Omron CX-Programmer project IO_TEST (CX-Programmer 9.20)

# PLC ELT215PLC: C200HE CPU42

## Global symbols (name address type ; comment)
0.00 BOOL  ; T_OUTPUT_FRONT GATE CLOSE
0.01 BOOL  ; T_OUTPUT_PULL IN PART
0.02 BOOL  ; T_OUTPUT_CLAMP ENGAGE
0.03 BOOL  ; T_OUTPUT_ALIGNMENT CLAMP RETRACT
0.04 BOOL  ; T_OUTPUT_TURNTABLE ROTATE FORWARD
0.05 BOOL  ; T_OUTPUT_EXIT GATE OPEN
0.06 BOOL  ; T_OUTPUT_DC_TEST_OUT
0.07 BOOL  ; T_OUTPUT_START SEQUENCER
0.08 BOOL  ; T_OUTPUT_BUZZER (INTERMITTENT)
0.09 BOOL  ; T_OUTPUT_PUSH OUT PART
0.10 BOOL  ; F_OUTPUT_FEED1 EXTEND
0.11 BOOL  ; F_OUTPUT_FEED2 EXTEND
0.12 BOOL  ; --== DO NOT USE ==--
0.13 BOOL  ; --== DO NOT USE ==--
0.14 BOOL  ; --== DO NOT USE ==--
0.15 BOOL  ; --== DO NOT USE ==--
1.00 BOOL  ; T_OUTPUT_THIRD TIME RELAY
1.01 BOOL  ; ID_OUTPUT_FRONT GATE CLOSE
1.02 BOOL  ; ID_OUTPUT_PUSH IN
1.03 BOOL  ; ID_OUTPUT_CLAMP ENGAGE
1.04 BOOL  ; ID_OUTPUT_TRAP DOOR OPEN
1.05 BOOL  ; ID_OUTPUT_PUSH OUT AND ELEVATE AND BACK GATE OPEN
1.06 BOOL  ; Output #6, Block 2 UNUSED
1.07 BOOL  ; ID_OUTPUT_JURASSIC GATE PULL UP
1.08 BOOL  ; --== DO NOT USE ==--
1.09 BOOL  ; --== DO NOT USE ==--
1.10 BOOL  ; --== DO NOT USE ==--
1.11 BOOL  ; --== DO NOT USE ==--
1.12 BOOL  ; --== DO NOT USE ==--
1.13 BOOL  ; --== DO NOT USE ==--
1.14 BOOL  ; --== DO NOT USE ==--
1.15 BOOL  ; --== DO NOT USE ==--
232.00 BOOL  ; F_WB_FEED1 EXTEND ONESHOT
232.01 BOOL  ; F_WB_FEED2 EXTEND ONESHOT
232.02 BOOL  ; F_WB_SEQUENCE RUNNING LATCH
232.03 BOOL  ; F_WB_FEEDER 1 PARTS EXTENSION PULSES
232.04 BOOL  ; F_WB_FEEDER 2 PARTS EXTENSION PULSES
232.05 BOOL  ; F_UNUSED WORK BIT
232.06 BOOL  ; F_UNUSED WORK BIT
232.07 BOOL  ; F_UNUSED WORK BIT
232.08 BOOL  ; F_UNUSED WORK BIT
232.09 BOOL  ; F_UNUSED WORK BIT
232.10 BOOL  ; F_UNUSED WORK BIT
232.11 BOOL  ; F_UNUSED WORK BIT
232.12 BOOL  ; F_UNUSED WORK BIT
232.13 BOOL  ; F_UNUSED WORK BIT
232.14 BOOL  ; F_UNUSED WORK BIT
232.15 BOOL  ; F_UNUSED WORK BIT
233.00 BOOL  ; F_UNUSED WORK BIT
233.01 BOOL  ; F_WB_PART 1 TIMER SILENCER
233.02 BOOL  ; F_WB_PART 2 TIMER SILENCER
233.03 BOOL  ; F_WB_PART 3 TIMER SILENCER
233.04 BOOL  ; F_WB_PART 4 TIMER SILENCER
233.05 BOOL  ; F_WB_PART 5 TIMER SILENCER
233.06 BOOL  ; F_WB_PART 6 TIMER SILENCER
233.07 BOOL  ; F_WB_PART 7 TIMER SILENCER
233.08 BOOL  ; F_WB_PART 8 TIMER SILENCER
233.09 BOOL  ; F_WB_PART 9 TIMER SILENCER
233.10 BOOL  ; F_WB_PART 10 TIMER SILENCER
233.11 BOOL  ; F_UNUSED WORK BIT
233.12 BOOL  ; F_UNUSED WORK BIT
233.13 BOOL  ; F_UNUSED WORK BIT
233.14 BOOL  ; F_UNUSED WORK BIT
233.15 BOOL  ; F_UNUSED WORK BIT
234.00 BOOL  ; F_UNUSED WORK BIT
234.01 BOOL  ; F_UNUSED WORK BIT
234.02 BOOL  ; F_UNUSED WORK BIT
234.03 BOOL  ; F_UNUSED WORK BIT
234.04 BOOL  ; F_UNUSED WORK BIT
234.05 BOOL  ; F_UNUSED WORK BIT
234.06 BOOL  ; F_UNUSED WORK BIT
234.07 BOOL  ; F_UNUSED WORK BIT
234.08 BOOL  ; F_UNUSED WORK BIT
234.09 BOOL  ; F_UNUSED WORK BIT
234.10 BOOL  ; F_UNUSED WORK BIT
234.11 BOOL  ; F_UNUSED WORK BIT
234.12 BOOL  ; F_UNUSED WORK BIT
234.13 BOOL  ; F_UNUSED WORK BIT
234.14 BOOL  ; F_UNUSED WORK BIT
234.15 BOOL  ; F_UNUSED WORK BIT
235.00 BOOL  ; F_UNUSED WORK BIT
235.01 BOOL  ; F_UNUSED WORK BIT
235.02 BOOL  ; F_UNUSED WORK BIT
235.03 BOOL  ; F_UNUSED WORK BIT
235.04 BOOL  ; F_UNUSED WORK BIT
235.05 BOOL  ; F_UNUSED WORK BIT
235.06 BOOL  ; F_UNUSED WORK BIT
235.07 BOOL  ; F_UNUSED WORK BIT
235.08 BOOL  ; F_UNUSED WORK BIT
235.09 BOOL  ; F_UNUSED WORK BIT
235.10 BOOL  ; F_UNUSED WORK BIT
235.11 BOOL  ; F_UNUSED WORK BIT
235.12 BOOL  ; F_UNUSED WORK BIT
235.13 BOOL  ; F_UNUSED WORK BIT
235.14 BOOL  ; F_UNUSED WORK BIT
235.15 BOOL  ; F_UNUSED WORK BIT
2.00 BOOL  ; T_INPUT_HSS
2.01 BOOL  ; T_INPUT_LSS
2.02 BOOL  ; T_INPUT_PAG SENSOR
2.03 BOOL  ; T_INPUT_TESTING STATION EMERGENCY HOME
2.04 BOOL  ; Input #4 Block 3
2.05 BOOL  ; ALL_INPUT_EMERGENCY HOME
2.06 BOOL  ; Input #6 Block 3
2.07 BOOL  ; F_INPUT_START FEEDER SEQUENCE
2.08 BOOL  ; F_INPUT_STOP FEEDER SEQUENCE
2.09 BOOL  ; Input #9 Block 3
2.10 BOOL  ; ID_INPUT_ID STATION EMERGENCY HOME
2.11 BOOL  ; ID_INPUT_IR PROXIMITY SENSOR
2.12 BOOL  ; ID_INPUT_THRU BEAM SENSOR
2.13 BOOL  ; ID_INPUT_ULTRASONIC SENSOR
2.14 BOOL  ; ID_INPUT_INDUCTIVE SENSOR
2.15 BOOL  ; ID_INPUT_PPG SENSOR
310.00 BOOL  ; T_WB_NEED HOLD FOR TESTING 1
310.01 BOOL  ; T_WB_NEED TO REORIENT 1
310.02 BOOL  ; T_NEED TO ABORT 1
310.03 BOOL  ; T_WB_NEED HOLD FOR TESTING 2
310.04 BOOL  ; T_WB_NEED TO REORIENT 2
310.05 BOOL  ; T_WB_NEED TO ABORT 2
310.06 BOOL  ; T_WB_LOCKED FRONT GATE CYLINDER LATCH
310.07 BOOL  ; T_WB_NEW PART AT GATE ONESHOT
310.08 BOOL  ; T_WB_NEW PAG DELAYED ONESHOT
310.09 BOOL  ; T_WB_PULL IN PART TRIG
310.10 BOOL  ; T_WB_LOCK FRONT GATE TRIG
310.11 BOOL  ; T_WB_RESEAT PART TRIG
310.12 BOOL  ; T_PULL IN TIMING ONESHOT
310.13 BOOL  ; T_WB_UNLOCK FRONT GATE TRIG
310.14 BOOL  ; T_WB_SEQ START PULSE
310.15 BOOL  ; T_WB_SEQ START DELAY LATCH
311.00 BOOL  ; T_WB_ABORT PROGRAM TRIG
311.01 BOOL  ; T_WB_T104 DRIVER
311.02 BOOL  ; T_WB_PART IN STATION LATCH
311.03 BOOL  ; T_WB_UNCLAMP
311.04 BOOL  ; T_WB_CLAMP
311.05 BOOL  ; T_WB_CLAMPED
311.06 BOOL  ; T_WB_ABORTING
311.07 BOOL  ; T_WB_REORIENTING
311.08 BOOL  ; T_WB_HOLDING FOR TEST
311.09 BOOL  ; T_WB_REORIENT DONE
311.10 BOOL  ; T_WB_ROTATE FORWARD DONE
311.11 BOOL  ; T_WB_ROTATE FORWARD WORKBIT
311.12 BOOL  ; T_WB_BUZZER ANNOUNCEMENT STATE
311.13 BOOL  ; T_WB_REORIENT UNCLAMP LENGTH PULSE
311.14 BOOL  ; T_WB_RESEATING PUSH DONE
311.15 BOOL  ; T_WB_RETRACT ALIGNMENT CLAMP
312.00 BOOL  ; T_WB_BACKWARDS ROTATION COMPLETE
312.01 BOOL  ; T_WB_LED TESTING STATE
312.02 BOOL  ; T_WB_DONE WITH TEST
312.03 BOOL  ; T_WB_DONE WITH TEST UNCLAMP PULSE LENGTH
312.04 BOOL  ; T_WB_READY FOR PUSH OUT
312.05 BOOL  ; T_WB_PUSHING OUT
312.06 BOOL  ; T_WB_OPEN EXIT GATE
312.07 BOOL  ; T_WB_T117 DRIVER
312.08 BOOL  ; T_WB_PLACEHOLDER
312.09 BOOL  ; T_WB_USED TO BE 0dot01 PULL IN PART
312.10 BOOL  ; T_WB_INITITAL PULL COMMAND LATCH
312.11 BOOL  ; T_WB_RESEAT PULL LATCH
312.12 BOOL  ; T_WB_USED TO BE PULL IN PART TRIG 310dot09
312.13 BOOL  ; T_WB_USED TO BE RESEAT PART TRIG 310dot11
312.14 BOOL  ; T_UNUSED WORK BIT
312.15 BOOL  ; T_UNUSED WORK BIT
313.00 BOOL  ; T_UNUSED WORK BIT
313.01 BOOL  ; T_UNUSED WORK BIT
313.02 BOOL  ; T_UNUSED WORK BIT
313.03 BOOL  ; T_UNUSED WORK BIT
313.04 BOOL  ; T_UNUSED WORK BIT
313.05 BOOL  ; T_UNUSED WORK BIT
313.06 BOOL  ; T_UNUSED WORK BIT
313.07 BOOL  ; T_UNUSED WORK BIT
313.08 BOOL  ; T_UNUSED WORK BIT
313.09 BOOL  ; T_UNUSED WORK BIT
313.10 BOOL  ; T_UNUSED WORK BIT
313.11 BOOL  ; T_UNUSED WORK BIT
313.12 BOOL  ; T_UNUSED WORK BIT
313.13 BOOL  ; T_UNUSED WORK BIT
313.14 BOOL  ; T_UNUSED WORK BIT
313.15 BOOL  ; T_UNUSED WORK BIT
314.00 BOOL  ; T_UNUSED WORK BIT
314.01 BOOL  ; T_UNUSED WORK BIT
314.02 BOOL  ; T_UNUSED WORK BIT
314.03 BOOL  ; T_UNUSED WORK BIT
314.04 BOOL  ; T_UNUSED WORK BIT
314.05 BOOL  ; T_UNUSED WORK BIT
314.06 BOOL  ; T_UNUSED WORK BIT
314.07 BOOL  ; T_UNUSED WORK BIT
314.08 BOOL  ; T_UNUSED WORK BIT
314.09 BOOL  ; T_UNUSED WORK BIT
314.10 BOOL  ; T_UNUSED WORK BIT
314.11 BOOL  ; T_UNUSED WORK BIT
314.12 BOOL  ; T_UNUSED WORK BIT
314.13 BOOL  ; T_UNUSED WORK BIT
314.14 BOOL  ; T_UNUSED WORK BIT
314.15 BOOL  ; T_UNUSED WORK BIT
315.00 BOOL  ; T_UNUSED WORK BIT
315.01 BOOL  ; T_UNUSED WORK BIT
315.02 BOOL  ; T_UNUSED WORK BIT
315.03 BOOL  ; T_UNUSED WORK BIT
315.04 BOOL  ; T_UNUSED WORK BIT
315.05 BOOL  ; T_UNUSED WORK BIT
315.06 BOOL  ; T_UNUSED WORK BIT
315.07 BOOL  ; T_UNUSED WORK BIT
315.08 BOOL  ; T_UNUSED WORK BIT
315.09 BOOL  ; T_UNUSED WORK BIT
315.10 BOOL  ; T_UNUSED WORK BIT
315.11 BOOL  ; T_UNUSED WORK BIT
315.12 BOOL  ; T_UNUSED WORK BIT
315.13 BOOL  ; T_UNUSED WORK BIT
315.14 BOOL  ; T_UNUSED WORK BIT
315.15 BOOL  ; T_UNUSED WORK BIT
316.00 BOOL  ; T_UNUSED WORK BIT
316.01 BOOL  ; T_UNUSED WORK BIT
316.02 BOOL  ; T_UNUSED WORK BIT
316.03 BOOL  ; T_UNUSED WORK BIT
316.04 BOOL  ; T_UNUSED WORK BIT
316.05 BOOL  ; T_UNUSED WORK BIT
316.06 BOOL  ; T_UNUSED WORK BIT
316.07 BOOL  ; T_UNUSED WORK BIT
316.08 BOOL  ; T_UNUSED WORK BIT
316.09 BOOL  ; T_UNUSED WORK BIT
316.10 BOOL  ; T_UNUSED WORK BIT
316.11 BOOL  ; T_UNUSED WORK BIT
316.12 BOOL  ; T_UNUSED WORK BIT
316.13 BOOL  ; T_UNUSED WORK BIT
316.14 BOOL  ; T_UNUSED WORK BIT
316.15 BOOL  ; T_UNUSED WORK BIT
317.00 BOOL  ; T_UNUSED WORK BIT
317.01 BOOL  ; T_UNUSED WORK BIT
317.02 BOOL  ; T_UNUSED WORK BIT
317.03 BOOL  ; T_UNUSED WORK BIT
317.04 BOOL  ; T_UNUSED WORK BIT
317.05 BOOL  ; T_UNUSED WORK BIT
317.06 BOOL  ; T_UNUSED WORK BIT
317.07 BOOL  ; T_UNUSED WORK BIT
317.08 BOOL  ; T_UNUSED WORK BIT
317.09 BOOL  ; T_UNUSED WORK BIT
317.10 BOOL  ; T_UNUSED WORK BIT
317.11 BOOL  ; T_UNUSED WORK BIT
317.12 BOOL  ; T_UNUSED WORK BIT
317.13 BOOL  ; T_UNUSED WORK BIT
317.14 BOOL  ; T_UNUSED WORK BIT
317.15 BOOL  ; T_UNUSED WORK BIT
318.00 BOOL  ; T_UNUSED WORK BIT
318.01 BOOL  ; T_UNUSED WORK BIT
318.02 BOOL  ; T_UNUSED WORK BIT
318.03 BOOL  ; T_UNUSED WORK BIT
318.04 BOOL  ; T_UNUSED WORK BIT
318.05 BOOL  ; T_UNUSED WORK BIT
318.06 BOOL  ; T_UNUSED WORK BIT
318.07 BOOL  ; T_UNUSED WORK BIT
318.08 BOOL  ; T_UNUSED WORK BIT
318.09 BOOL  ; T_UNUSED WORK BIT
318.10 BOOL  ; T_UNUSED WORK BIT
318.11 BOOL  ; T_UNUSED WORK BIT
318.12 BOOL  ; T_UNUSED WORK BIT
318.13 BOOL  ; T_UNUSED WORK BIT
318.14 BOOL  ; T_UNUSED WORK BIT
318.15 BOOL  ; T_UNUSED WORK BIT
319.00 BOOL  ; T_UNUSED WORK BIT
319.01 BOOL  ; T_UNUSED WORK BIT
319.02 BOOL  ; T_UNUSED WORK BIT
319.03 BOOL  ; T_UNUSED WORK BIT
319.04 BOOL  ; T_UNUSED WORK BIT
319.05 BOOL  ; T_UNUSED WORK BIT
319.06 BOOL  ; T_UNUSED WORK BIT
319.07 BOOL  ; T_UNUSED WORK BIT
319.08 BOOL  ; T_UNUSED WORK BIT
319.09 BOOL  ; T_UNUSED WORK BIT
319.10 BOOL  ; T_UNUSED WORK BIT
319.11 BOOL  ; T_UNUSED WORK BIT
319.12 BOOL  ; T_UNUSED WORK BIT
319.13 BOOL  ; T_UNUSED WORK BIT
319.14 BOOL  ; T_UNUSED WORK BIT
319.15 BOOL  ; T_UNUSED WORK BIT
320.00 BOOL  ; ID_WB_3 SENSOR METHOD
320.01 BOOL  ; ID_WB_4 SENSOR METHOD
320.02 BOOL  ; ID_WB_REJECT PART PRESENT
320.03 BOOL  ; ID_WB_SMALL PART PRESENT
320.04 BOOL  ; ID_WB_ELECTRONIC PART PRESENT
320.05 BOOL  ; ID_WB_LARGE PART PRESENT
320.06 BOOL  ; ID_WB_NO PART PRESENT
320.07 BOOL  ; ID_WB_UNKNOWN PART PRESENT
320.08 BOOL  ; ID_WB_NEED TO OPEN TRAP DOOR 1
320.09 BOOL  ; ID_WB_NEED TO PUSH OUT WITH JURASSIC CLOSED 1
320.10 BOOL  ; ID_WB_NEED TO PUSH OUT WITH JURASSIC OPEN 1
320.11 BOOL  ; ID_WB_NEED TO RESET 1
320.12 BOOL  ; ID_WB_LOCKED FRONT GATE LATCH
320.13 BOOL  ; ID_WB_LOCK FRONT GATE TRIGGER
320.14 BOOL  ; ID_WB_UNLOCK FRONT GATE TIMER LATCH
320.15 BOOL  ; ID_WB_PART IS AT CLOSED EXIT GATE
321.00 BOOL  ; ID_WB_PART IS UNCLAMPED BUT IN SCANNING AREA
321.01 BOOL  ; ID_WB_PUSH IN PART COMMAND WORKBIT
321.02 BOOL  ; ID_WB_WAITING FOR PUSHER TO GET OUT ONE SHOT
321.03 BOOL  ; ID_WB_CLAMPED
321.04 BOOL  ; ID_WB_CLAMPING
321.05 BOOL  ; ID_WB_UNCLAMP LATCH
321.06 BOOL  ; ID_WB_UNCLAMPED
321.07 BOOL  ; ID_WB_UNCLAMP TRIGGER FROM REJECT
321.08 BOOL  ; ID_WB_NEED TO OPEN TRAP DOOR 2
321.09 BOOL  ; ID_WB_NEED TO PUSH OUT WITH JURASSIC CLOSED 2
321.10 BOOL  ; ID_WB_NEED TO PUSH OUT WITH JURASSIC OPEN 2
321.11 BOOL  ; ID_WB_NEED TO RESET 2
321.12 BOOL  ; ID_WB_SYSTEM RESET ONESHOT
321.13 BOOL  ; ID_WB_UNLOCK FRONT GATE TRIGGER
321.14 BOOL  ; ID_WB_PUSH RETRACTION TIMING LATCH
321.15 BOOL  ; ID_WB_SEQUENCE COMPLETE 2
322.00 BOOL  ; ID_WB_SEQUENCE COMPLETE 1
322.01 BOOL  ; ID_WB_REJECT SEQUENCE RUNNING LATCH
322.02 BOOL  ; ID_WB_PUSH OUT TRIGGER FOR UNKNOWN
322.03 BOOL  ; ID_WB_PUSH OUT LATCH
322.04 BOOL  ; ID_WB_SYSTEM RESET LATCH
322.05 BOOL  ; ID_WB PUSH OUT TRIGGER FOR SMALL
322.06 BOOL  ; ID_WB_PUSH OUT TRIGGER FOR LARGE
322.07 BOOL  ; ID_WB PUSH OUT TRIGGER FOR ELECTRONIC
322.08 BOOL  ; ID_WB_SMALL LARGE UNKNOWN SEQUENCE RUNNING LATCH
322.09 BOOL  ; ID_WB_ELECTRONIC PART SEQUENCE RUNNING LATCH
322.10 BOOL  ; ID_WB_RAISE JURASSIC GATE
322.11 BOOL  ; ID_TRAP DOOR OPEN ENDING EDGE LATCH
322.12 BOOL  ; ID_RESET REQUEST
322.13 BOOL  ; ID_WB_UNCLAMP TRIGGER FROM SMALL LARGE UNKNOWN
322.14 BOOL  ; ID_WB_UNCLAMP TRIGGER FROM ELECTRONIC
322.15 BOOL  ; ID_WB_JURASSIC GATE RAISED
323.00 BOOL  ; ID_WB_PUSHING IN IS DONE UNTIL NEXT TEST
323.01 BOOL  ; ID_WB_CLAMPING IS DONE UNTIL NEXT TEST
323.02 BOOL  ; ID_WB_PLACEHOLDER
323.03 BOOL  ; ID_UNUSED WORK BIT
323.04 BOOL  ; ID_UNUSED WORK BIT
323.05 BOOL  ; ID_UNUSED WORK BIT
323.06 BOOL  ; ID_UNUSED WORK BIT
323.07 BOOL  ; ID_UNUSED WORK BIT
323.08 BOOL  ; ID_UNUSED WORK BIT
323.09 BOOL  ; ID_UNUSED WORK BIT
323.10 BOOL  ; ID_UNUSED WORK BIT
323.11 BOOL  ; ID_UNUSED WORK BIT
323.12 BOOL  ; ID_UNUSED WORK BIT
323.13 BOOL  ; ID_UNUSED WORK BIT
323.14 BOOL  ; ID_UNUSED WORK BIT
323.15 BOOL  ; ID_UNUSED WORK BIT
324.00 BOOL  ; ID_UNUSED WORK BIT
324.01 BOOL  ; ID_UNUSED WORK BIT
324.02 BOOL  ; ID_UNUSED WORK BIT
324.03 BOOL  ; ID_UNUSED WORK BIT
324.04 BOOL  ; ID_UNUSED WORK BIT
324.05 BOOL  ; ID_UNUSED WORK BIT
324.06 BOOL  ; ID_UNUSED WORK BIT
324.07 BOOL  ; ID_UNUSED WORK BIT
324.08 BOOL  ; ID_UNUSED WORK BIT
324.09 BOOL  ; ID_UNUSED WORK BIT
324.10 BOOL  ; ID_UNUSED WORK BIT
324.11 BOOL  ; ID_UNUSED WORK BIT
324.12 BOOL  ; ID_UNUSED WORK BIT
324.13 BOOL  ; ID_UNUSED WORK BIT
324.14 BOOL  ; ID_UNUSED WORK BIT
324.15 BOOL  ; ID_UNUSED WORK BIT
325.00 BOOL  ; ID_UNUSED WORK BIT
325.01 BOOL  ; ID_UNUSED WORK BIT
325.02 BOOL  ; ID_UNUSED WORK BIT
325.03 BOOL  ; ID_UNUSED WORK BIT
325.04 BOOL  ; ID_UNUSED WORK BIT
325.05 BOOL  ; ID_UNUSED WORK BIT
325.06 BOOL  ; ID_UNUSED WORK BIT
325.07 BOOL  ; ID_UNUSED WORK BIT
325.08 BOOL  ; ID_UNUSED WORK BIT
325.09 BOOL  ; ID_UNUSED WORK BIT
325.10 BOOL  ; ID_UNUSED WORK BIT
325.11 BOOL  ; ID_UNUSED WORK BIT
325.12 BOOL  ; ID_UNUSED WORK BIT
325.13 BOOL  ; ID_UNUSED WORK BIT
325.14 BOOL  ; ID_UNUSED WORK BIT
325.15 BOOL  ; ID_UNUSED WORK BIT
326.00 BOOL  ; ID_UNUSED WORK BIT
326.01 BOOL  ; ID_UNUSED WORK BIT
326.02 BOOL  ; ID_UNUSED WORK BIT
326.03 BOOL  ; ID_UNUSED WORK BIT
326.04 BOOL  ; ID_UNUSED WORK BIT
326.05 BOOL  ; ID_UNUSED WORK BIT
326.06 BOOL  ; ID_UNUSED WORK BIT
326.07 BOOL  ; ID_UNUSED WORK BIT
326.08 BOOL  ; ID_UNUSED WORK BIT
326.09 BOOL  ; ID_UNUSED WORK BIT
326.10 BOOL  ; ID_UNUSED WORK BIT
326.11 BOOL  ; ID_UNUSED WORK BIT
326.12 BOOL  ; ID_UNUSED WORK BIT
326.13 BOOL  ; ID_UNUSED WORK BIT
326.14 BOOL  ; ID_UNUSED WORK BIT
326.15 BOOL  ; ID_UNUSED WORK BIT
327.00 BOOL  ; ID_UNUSED WORK BIT
327.01 BOOL  ; ID_UNUSED WORK BIT
327.02 BOOL  ; ID_UNUSED WORK BIT
327.03 BOOL  ; ID_UNUSED WORK BIT
327.04 BOOL  ; ID_UNUSED WORK BIT
327.05 BOOL  ; ID_UNUSED WORK BIT
327.06 BOOL  ; ID_UNUSED WORK BIT
327.07 BOOL  ; ID_UNUSED WORK BIT
327.08 BOOL  ; ID_UNUSED WORK BIT
327.09 BOOL  ; ID_UNUSED WORK BIT
327.10 BOOL  ; ID_UNUSED WORK BIT
327.11 BOOL  ; ID_UNUSED WORK BIT
327.12 BOOL  ; ID_UNUSED WORK BIT
327.13 BOOL  ; ID_UNUSED WORK BIT
327.14 BOOL  ; ID_UNUSED WORK BIT
327.15 BOOL  ; ID_UNUSED WORK BIT
328.00 BOOL  ; ID_UNUSED WORK BIT
328.01 BOOL  ; ID_UNUSED WORK BIT
328.02 BOOL  ; ID_UNUSED WORK BIT
328.03 BOOL  ; ID_UNUSED WORK BIT
328.04 BOOL  ; ID_UNUSED WORK BIT
328.05 BOOL  ; ID_UNUSED WORK BIT
328.06 BOOL  ; ID_UNUSED WORK BIT
328.07 BOOL  ; ID_UNUSED WORK BIT
328.08 BOOL  ; ID_UNUSED WORK BIT
328.09 BOOL  ; ID_UNUSED WORK BIT
328.10 BOOL  ; ID_UNUSED WORK BIT
328.11 BOOL  ; ID_UNUSED WORK BIT
328.12 BOOL  ; ID_UNUSED WORK BIT
328.13 BOOL  ; ID_UNUSED WORK BIT
328.14 BOOL  ; ID_UNUSED WORK BIT
328.15 BOOL  ; ID_UNUSED WORK BIT
329.00 BOOL  ; ID_UNUSED WORK BIT
329.01 BOOL  ; ID_UNUSED WORK BIT
329.02 BOOL  ; ID_UNUSED WORK BIT
329.03 BOOL  ; ID_UNUSED WORK BIT
329.04 BOOL  ; ID_UNUSED WORK BIT
329.05 BOOL  ; ID_UNUSED WORK BIT
329.06 BOOL  ; ID_UNUSED WORK BIT
329.07 BOOL  ; ID_UNUSED WORK BIT
329.08 BOOL  ; ID_UNUSED WORK BIT
329.09 BOOL  ; ID_UNUSED WORK BIT
329.10 BOOL  ; ID_UNUSED WORK BIT
329.11 BOOL  ; ID_UNUSED WORK BIT
329.12 BOOL  ; ID_UNUSED WORK BIT
329.13 BOOL  ; ID_UNUSED WORK BIT
329.14 BOOL  ; ID_UNUSED WORK BIT
329.15 BOOL  ; ID_UNUSED WORK BIT
CNT511 BOOL  ; T_THIRD TIME COUNTER
TIM000 BOOL  ; ID_PART ARRIVAL DELAY
TIM001 BOOL  ; ID_PUSH IN PART ONE SHOT LENGTH
TIM002 BOOL  ; ID_PUSHER GETTING OUT ONE SHOT LENGTH
TIM003 BOOL  ; ID_TIME TO CLAMP
TIM004 BOOL  ; ID_TIME TO UNCLAMP
TIM005 BOOL  ; ID_WAIT TO OPEN FRONT GATE UPON RESET
TIM006 BOOL  ; ID_WAIT FOR PUSH AND ELEVATE CYLINDERS TO RETRACT BEFORE SYSTEM RESET
TIM007 BOOL  ; ID_PUSH OUT TIMING
TIM008 BOOL  ; ID_LENGTH OF SYSTEM RESET ONESHOT
TIM009 BOOL  ; ID_LENGTH UNTIL SYSTEM RESET, WHICH CLOSES TRAP DOOR
TIM010 BOOL  ; ID_TIME FOR JURASSIC GATE TO OPEN
TIM100 BOOL  ; T_PULL IN TIMING ONESHOT
TIM101 BOOL  ; T_NEW PART AT GATE ONESHOT
TIM102 BOOL  ; T_NEW PART AT GATE ONESHOT DELAY
TIM103 BOOL  ; T_COLLISION AVOIDANCE DELAY FOR STATION 2 AND 3 COMPLETION
TIM104 BOOL  ; T_INITIAL PULL IN AND RETRACT TIMING
TIM105 BOOL  ; T_TIME IT TAKES TO CLAMP
TIM106 BOOL  ; T_LENGTH OF FORWARD ROTATE
TIM107 BOOL  ; T_TIME TO UNCLAMP ALL THREE
TIM108 BOOL  ; T_TIME TO ROTATE BACKWARDS
TIM109 BOOL  ; T_REORIENT DONE ONESHOT LENGTH
TIM110 BOOL  ; T_LENGTH OF BUZZER ANNOUNCEMENT STATE
TIM111 BOOL  ; T_LENGTH OF LED TESTING STATE
TIM112 BOOL  ; T_TIME TO UNCLAMP MAIN CLAMPS
TIM113 BOOL  ; T_TIME TO PUSH OUT
TIM114 BOOL  ; T_LENGTH OF EXIT GATE OPEN
TIM115 BOOL  ; T_DELAY UNTIL SEQ START
TIM116 BOOL  ; T_WIDTH OF SEQ START PULSE
TIM117 BOOL  ; T_RESEAT PULL IN AND RETRACT TIMING
TIM118 BOOL  ; T_PULL IN TIME FROM PULLING IN
TIM119 BOOL  ; T_PULL IN TIME FROM RESEAT
TIM200 BOOL  ; F_SEQUENCE OVER TIME
TIM201 BOOL  ; F_PART 1 TIME
TIM202 BOOL  ; F_PART 2 TIME
TIM203 BOOL  ; F_PART 3 TIME
TIM204 BOOL  ; F_PART 4 TIME
TIM205 BOOL  ; F_PART 5 TIME
TIM206 BOOL  ; F_PART 6 TIME
TIM207 BOOL  ; F_PART 7 TIME
TIM208 BOOL  ; F_PART 8 TIME
TIM209 BOOL  ; F_PART 9 TIME
TIM210 BOOL  ; F_PART 10 TIME
TIM301 BOOL  ; F_FEED 1 EXTENSION TIME
TIM302 BOOL  ; F_FEED 2 EXTENSION TIME

## Program ELT215_SPRING2012 (no task)
; 'PLC TO RUN:   "T" Electronic Part Testing Station        "ID" All 4 Part Identification Station           and "F" Feeder Sequencing'

### Section UNIVERSAL_PARAMETERS
; 'Parameters that control large changes in the ladder logic.  The "user editable" section to be changed on the fly.'

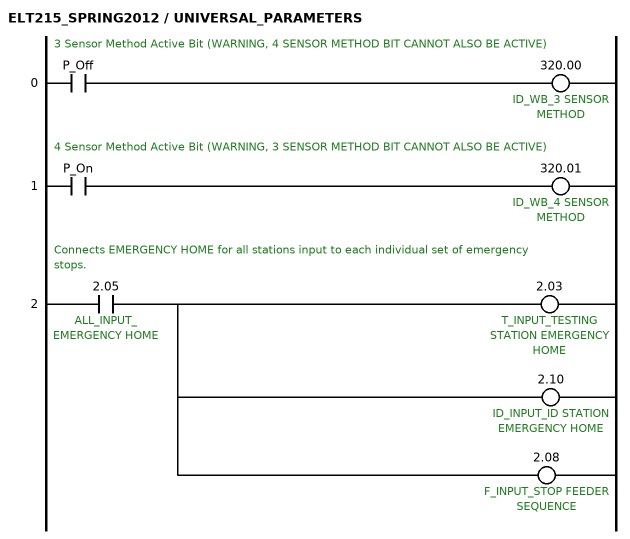
; rung 0: 3 Sensor Method Active Bit (WARNING, 4 SENSOR METHOD BIT CANNOT ALSO BE ACTIVE)
LD P_Off
OUT 320.00  ; ID_WB_3 SENSOR METHOD
; rung 1: 4 Sensor Method Active Bit (WARNING, 3 SENSOR METHOD BIT CANNOT ALSO BE ACTIVE)
LD P_On
OUT 320.01  ; ID_WB_4 SENSOR METHOD
; rung 2: Connects EMERGENCY HOME for all stations input to each individual set of emergency stops.
LD 2.05  ; ALL_INPUT_EMERGENCY HOME
OUT 2.03  ; T_INPUT_TESTING STATION EMERGENCY HOME
OUT 2.10  ; ID_INPUT_ID STATION EMERGENCY HOME
OUT 2.08  ; F_INPUT_STOP FEEDER SEQUENCE

### Section ID_GETTING_PART_TO_SCANNING_AREA
; Ladder logic for ID Station to identify a part has come in, prevent other parts from getting in, and clamp the part.

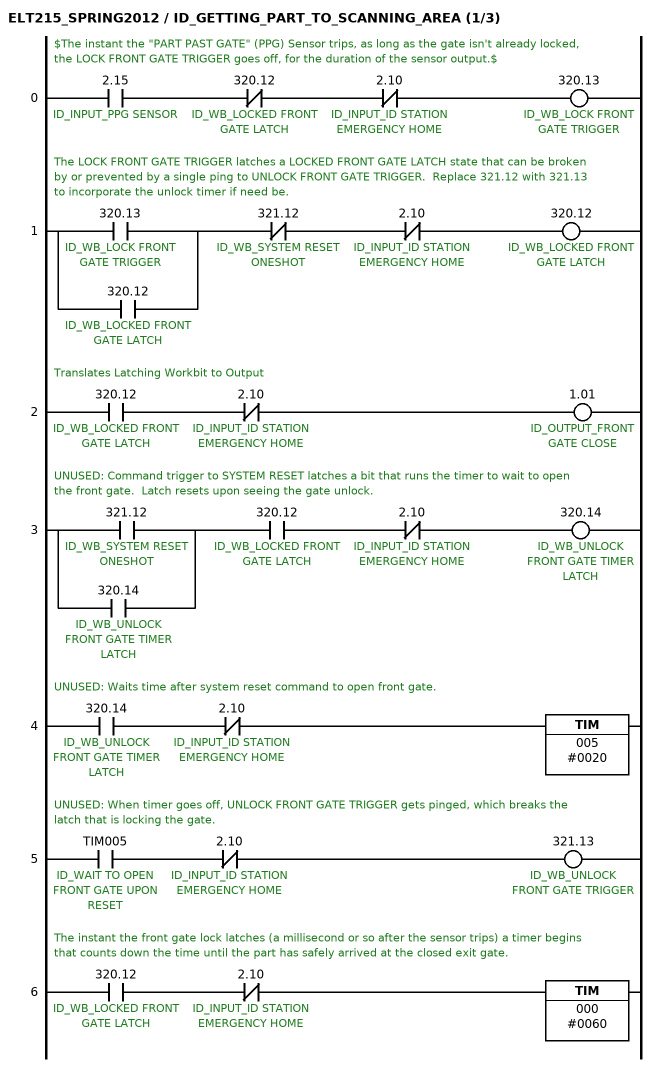
; rung 0: $The instant the "PART PAST GATE" (PPG) Sensor trips, as long as the gate isn't already locked, the LOCK FRONT GATE TRIGGER goes off, for the duration of the sensor output.$
LD 2.15  ; ID_INPUT_PPG SENSOR
ANDNOT 320.12  ; ID_WB_LOCKED FRONT GATE LATCH
ANDNOT 2.10  ; ID_INPUT_ID STATION EMERGENCY HOME
OUT 320.13  ; ID_WB_LOCK FRONT GATE TRIGGER
; rung 1: The LOCK FRONT GATE TRIGGER latches a LOCKED FRONT GATE LATCH state that can be broken by or prevented by a single ping to UNLOCK FRONT GATE TRIGGER.  Replace 321.12 with 321.13 to incorporate the unlock timer if need be.
LD 320.13  ; ID_WB_LOCK FRONT GATE TRIGGER
OR 320.12  ; ID_WB_LOCKED FRONT GATE LATCH
ANDNOT 321.12  ; ID_WB_SYSTEM RESET ONESHOT
ANDNOT 2.10  ; ID_INPUT_ID STATION EMERGENCY HOME
OUT 320.12  ; ID_WB_LOCKED FRONT GATE LATCH
; rung 2: Translates Latching Workbit to Output
LD 320.12  ; ID_WB_LOCKED FRONT GATE LATCH
ANDNOT 2.10  ; ID_INPUT_ID STATION EMERGENCY HOME
OUT 1.01  ; ID_OUTPUT_FRONT GATE CLOSE
; rung 3: UNUSED: Command trigger to SYSTEM RESET latches a bit that runs the timer to wait to open the front gate.  Latch resets upon seeing the gate unlock.
LD 321.12  ; ID_WB_SYSTEM RESET ONESHOT
OR 320.14  ; ID_WB_UNLOCK FRONT GATE TIMER LATCH
AND 320.12  ; ID_WB_LOCKED FRONT GATE LATCH
ANDNOT 2.10  ; ID_INPUT_ID STATION EMERGENCY HOME
OUT 320.14  ; ID_WB_UNLOCK FRONT GATE TIMER LATCH
; rung 4: UNUSED: Waits time after system reset command to open front gate.
LD 320.14  ; ID_WB_UNLOCK FRONT GATE TIMER LATCH
ANDNOT 2.10  ; ID_INPUT_ID STATION EMERGENCY HOME
TIM 005 #0020
; rung 5: UNUSED: When timer goes off, UNLOCK FRONT GATE TRIGGER gets pinged, which breaks the latch that is locking the gate.
LD TIM005  ; ID_WAIT TO OPEN FRONT GATE UPON RESET
ANDNOT 2.10  ; ID_INPUT_ID STATION EMERGENCY HOME
OUT 321.13  ; ID_WB_UNLOCK FRONT GATE TRIGGER
; rung 6: The instant the front gate lock latches (a millisecond or so after the sensor trips) a timer begins that counts down the time until the part has safely arrived at the closed exit gate.
LD 320.12  ; ID_WB_LOCKED FRONT GATE LATCH
ANDNOT 2.10  ; ID_INPUT_ID STATION EMERGENCY HOME
TIM 000 #0060

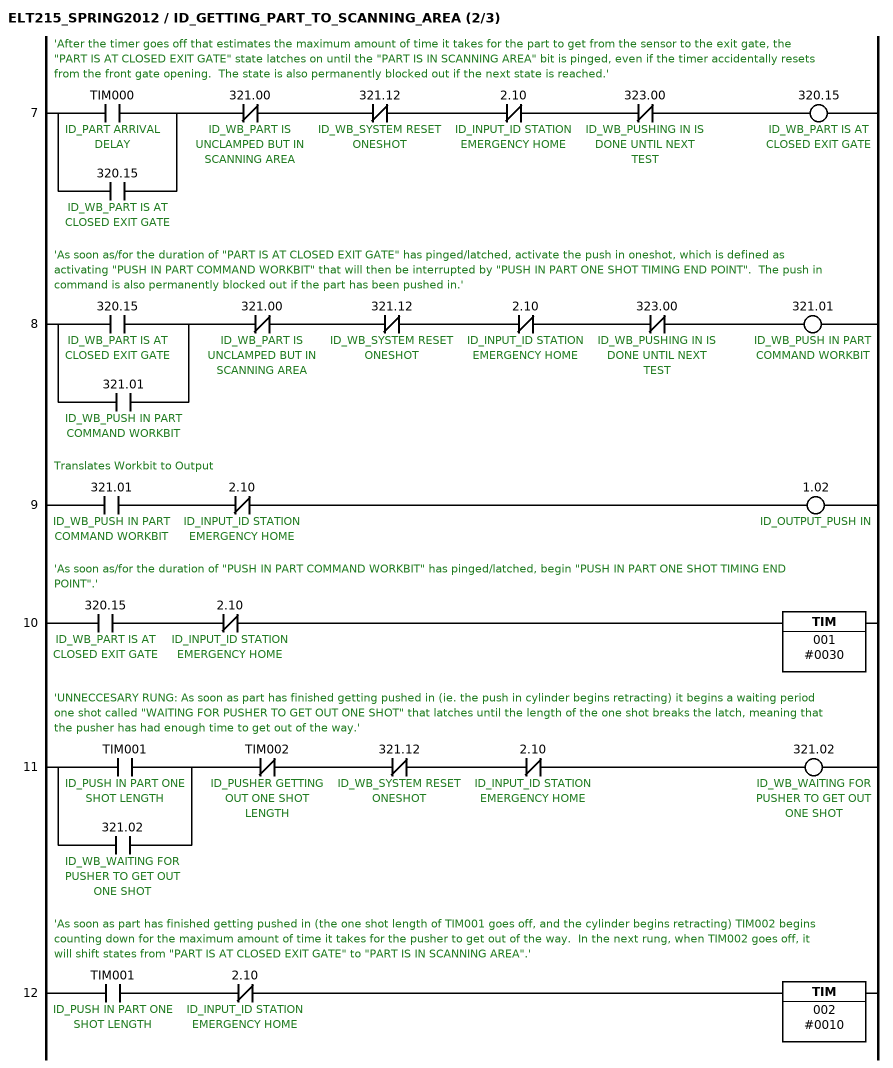
; rung 7: 'After the timer goes off that estimates the maximum amount of time it takes for the part to get from the sensor to the exit gate, the "PART IS AT CLOSED EXIT GATE" state latches on until the "PART IS IN SCANNING AREA" bit is pinged, even if the timer accidentally resets from the front gate opening.  The state is also permanently blocked out if the next state is reached.'
LD TIM000  ; ID_PART ARRIVAL DELAY
OR 320.15  ; ID_WB_PART IS AT CLOSED EXIT GATE
ANDNOT 321.00  ; ID_WB_PART IS UNCLAMPED BUT IN SCANNING AREA
ANDNOT 321.12  ; ID_WB_SYSTEM RESET ONESHOT
ANDNOT 2.10  ; ID_INPUT_ID STATION EMERGENCY HOME
ANDNOT 323.00  ; ID_WB_PUSHING IN IS DONE UNTIL NEXT TEST
OUT 320.15  ; ID_WB_PART IS AT CLOSED EXIT GATE
; rung 8: 'As soon as/for the duration of "PART IS AT CLOSED EXIT GATE" has pinged/latched, activate the push in oneshot, which is defined as activating "PUSH IN PART COMMAND WORKBIT" that will then be interrupted by "PUSH IN PART ONE SHOT TIMING END POINT".  The push in command is also permanently blocked out if the part has been pushed in.'
LD 320.15  ; ID_WB_PART IS AT CLOSED EXIT GATE
OR 321.01  ; ID_WB_PUSH IN PART COMMAND WORKBIT
ANDNOT 321.00  ; ID_WB_PART IS UNCLAMPED BUT IN SCANNING AREA
ANDNOT 321.12  ; ID_WB_SYSTEM RESET ONESHOT
ANDNOT 2.10  ; ID_INPUT_ID STATION EMERGENCY HOME
ANDNOT 323.00  ; ID_WB_PUSHING IN IS DONE UNTIL NEXT TEST
OUT 321.01  ; ID_WB_PUSH IN PART COMMAND WORKBIT
; rung 9: Translates Workbit to Output
LD 321.01  ; ID_WB_PUSH IN PART COMMAND WORKBIT
ANDNOT 2.10  ; ID_INPUT_ID STATION EMERGENCY HOME
OUT 1.02  ; ID_OUTPUT_PUSH IN
; rung 10: 'As soon as/for the duration of "PUSH IN PART COMMAND WORKBIT" has pinged/latched, begin "PUSH IN PART ONE SHOT TIMING END POINT".'
LD 320.15  ; ID_WB_PART IS AT CLOSED EXIT GATE
ANDNOT 2.10  ; ID_INPUT_ID STATION EMERGENCY HOME
TIM 001 #0030
; rung 11: 'UNNECCESARY RUNG: As soon as part has finished getting pushed in (ie. the push in cylinder begins retracting) it begins a waiting period one shot called "WAITING FOR PUSHER TO GET OUT ONE SHOT" that latches until the length of the one shot breaks the latch, meaning that the pusher has had enough time to get out of the way.'
LD TIM001  ; ID_PUSH IN PART ONE SHOT LENGTH
OR 321.02  ; ID_WB_WAITING FOR PUSHER TO GET OUT ONE SHOT
ANDNOT TIM002  ; ID_PUSHER GETTING OUT ONE SHOT LENGTH
ANDNOT 321.12  ; ID_WB_SYSTEM RESET ONESHOT
ANDNOT 2.10  ; ID_INPUT_ID STATION EMERGENCY HOME
OUT 321.02  ; ID_WB_WAITING FOR PUSHER TO GET OUT ONE SHOT
; rung 12: 'As soon as part has finished getting pushed in (the one shot length of TIM001 goes off, and the cylinder begins retracting) TIM002 begins counting down for the maximum amount of time it takes for the pusher to get out of the way.  In the next rung, when TIM002 goes off, it will shift states from "PART IS AT CLOSED EXIT GATE" to "PART IS IN SCANNING AREA".'
LD TIM001  ; ID_PUSH IN PART ONE SHOT LENGTH
ANDNOT 2.10  ; ID_INPUT_ID STATION EMERGENCY HOME
TIM 002 #0010

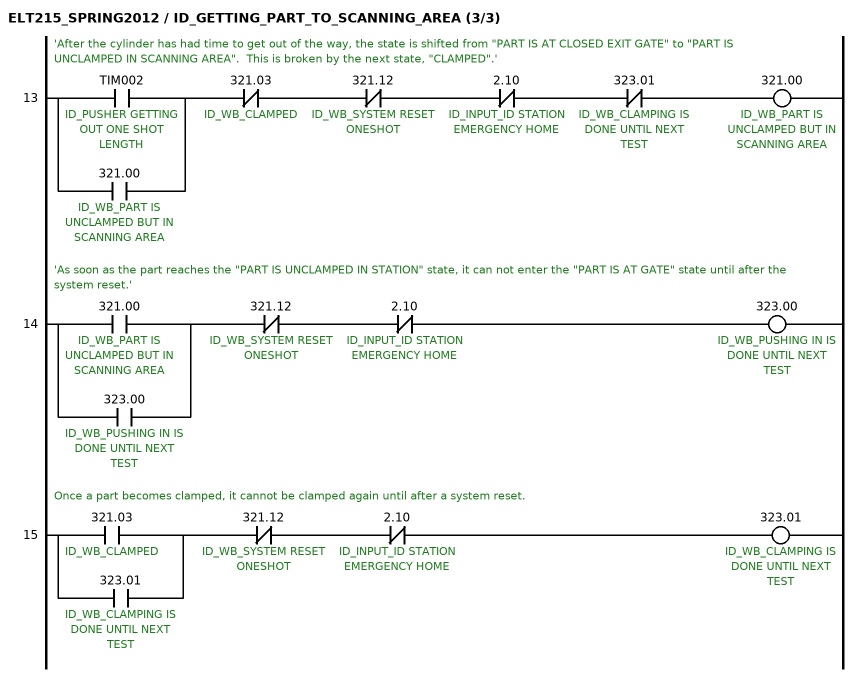
; rung 13: 'After the cylinder has had time to get out of the way, the state is shifted from "PART IS AT CLOSED EXIT GATE" to "PART IS UNCLAMPED IN SCANNING AREA".  This is broken by the next state, "CLAMPED".'
LD TIM002  ; ID_PUSHER GETTING OUT ONE SHOT LENGTH
OR 321.00  ; ID_WB_PART IS UNCLAMPED BUT IN SCANNING AREA
ANDNOT 321.03  ; ID_WB_CLAMPED
ANDNOT 321.12  ; ID_WB_SYSTEM RESET ONESHOT
ANDNOT 2.10  ; ID_INPUT_ID STATION EMERGENCY HOME
ANDNOT 323.01  ; ID_WB_CLAMPING IS DONE UNTIL NEXT TEST
OUT 321.00  ; ID_WB_PART IS UNCLAMPED BUT IN SCANNING AREA
; rung 14: 'As soon as the part reaches the "PART IS UNCLAMPED IN STATION" state, it can not enter the "PART IS AT GATE" state until after the system reset.'
LD 321.00  ; ID_WB_PART IS UNCLAMPED BUT IN SCANNING AREA
OR 323.00  ; ID_WB_PUSHING IN IS DONE UNTIL NEXT TEST
ANDNOT 321.12  ; ID_WB_SYSTEM RESET ONESHOT
ANDNOT 2.10  ; ID_INPUT_ID STATION EMERGENCY HOME
OUT 323.00  ; ID_WB_PUSHING IN IS DONE UNTIL NEXT TEST
; rung 15: Once a part becomes clamped, it cannot be clamped again until after a system reset.
LD 321.03  ; ID_WB_CLAMPED
OR 323.01  ; ID_WB_CLAMPING IS DONE UNTIL NEXT TEST
ANDNOT 321.12  ; ID_WB_SYSTEM RESET ONESHOT
ANDNOT 2.10  ; ID_INPUT_ID STATION EMERGENCY HOME
OUT 323.01  ; ID_WB_CLAMPING IS DONE UNTIL NEXT TEST

### Section ID_CLAMPING_AND_UNCLAMPING_PART
; Manages the CLAMPING, UNCLAMPING, CLAMPED, and UNCLAMPED states.

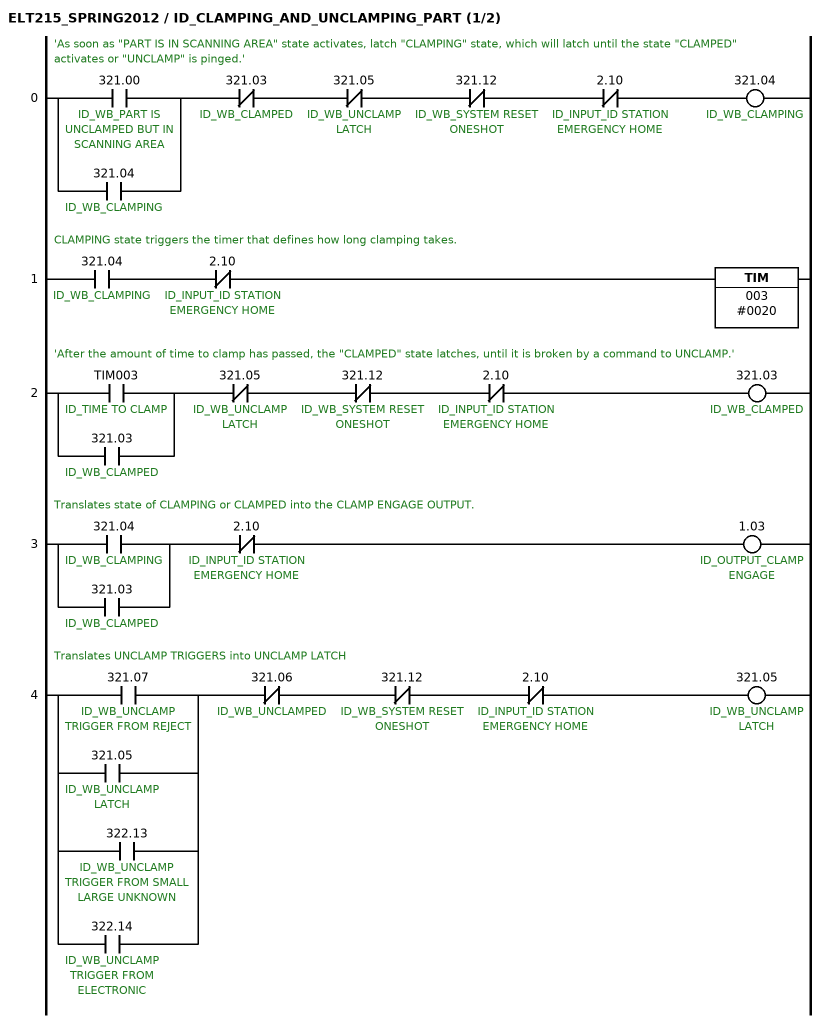
; rung 0: 'As soon as "PART IS IN SCANNING AREA" state activates, latch "CLAMPING" state, which will latch until the state "CLAMPED" activates or "UNCLAMP" is pinged.'
LD 321.00  ; ID_WB_PART IS UNCLAMPED BUT IN SCANNING AREA
OR 321.04  ; ID_WB_CLAMPING
ANDNOT 321.03  ; ID_WB_CLAMPED
ANDNOT 321.05  ; ID_WB_UNCLAMP LATCH
ANDNOT 321.12  ; ID_WB_SYSTEM RESET ONESHOT
ANDNOT 2.10  ; ID_INPUT_ID STATION EMERGENCY HOME
OUT 321.04  ; ID_WB_CLAMPING
; rung 1: CLAMPING state triggers the timer that defines how long clamping takes.
LD 321.04  ; ID_WB_CLAMPING
ANDNOT 2.10  ; ID_INPUT_ID STATION EMERGENCY HOME
TIM 003 #0020
; rung 2: 'After the amount of time to clamp has passed, the "CLAMPED" state latches, until it is broken by a command to UNCLAMP.'
LD TIM003  ; ID_TIME TO CLAMP
OR 321.03  ; ID_WB_CLAMPED
ANDNOT 321.05  ; ID_WB_UNCLAMP LATCH
ANDNOT 321.12  ; ID_WB_SYSTEM RESET ONESHOT
ANDNOT 2.10  ; ID_INPUT_ID STATION EMERGENCY HOME
OUT 321.03  ; ID_WB_CLAMPED
; rung 3: Translates state of CLAMPING or CLAMPED into the CLAMP ENGAGE OUTPUT.
LD 321.04  ; ID_WB_CLAMPING
OR 321.03  ; ID_WB_CLAMPED
ANDNOT 2.10  ; ID_INPUT_ID STATION EMERGENCY HOME
OUT 1.03  ; ID_OUTPUT_CLAMP ENGAGE
; rung 4: Translates UNCLAMP TRIGGERS into UNCLAMP LATCH
LD 321.07  ; ID_WB_UNCLAMP TRIGGER FROM REJECT
OR 321.05  ; ID_WB_UNCLAMP LATCH
OR 322.13  ; ID_WB_UNCLAMP TRIGGER FROM SMALL LARGE UNKNOWN
OR 322.14  ; ID_WB_UNCLAMP TRIGGER FROM ELECTRONIC
ANDNOT 321.06  ; ID_WB_UNCLAMPED
ANDNOT 321.12  ; ID_WB_SYSTEM RESET ONESHOT
ANDNOT 2.10  ; ID_INPUT_ID STATION EMERGENCY HOME
OUT 321.05  ; ID_WB_UNCLAMP LATCH

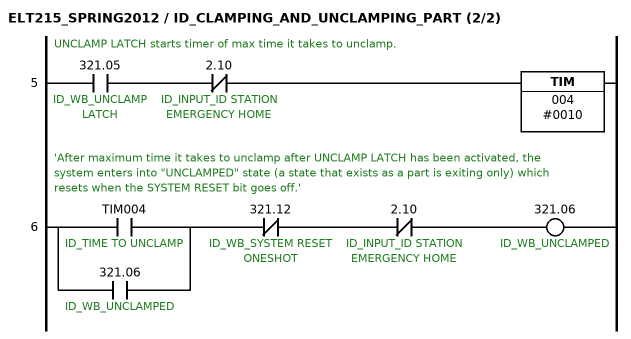
; rung 5: UNCLAMP LATCH starts timer of max time it takes to unclamp.
LD 321.05  ; ID_WB_UNCLAMP LATCH
ANDNOT 2.10  ; ID_INPUT_ID STATION EMERGENCY HOME
TIM 004 #0010
; rung 6: 'After maximum time it takes to unclamp after UNCLAMP LATCH has been activated, the system enters into "UNCLAMPED" state (a state that exists as a part is exiting only) which resets when the SYSTEM RESET bit goes off.'
LD TIM004  ; ID_TIME TO UNCLAMP
OR 321.06  ; ID_WB_UNCLAMPED
ANDNOT 321.12  ; ID_WB_SYSTEM RESET ONESHOT
ANDNOT 2.10  ; ID_INPUT_ID STATION EMERGENCY HOME
OUT 321.06  ; ID_WB_UNCLAMPED

### Section ID_IDENTIFICATION_MATRIX_AND_REQUESTS
; Combinational logic that converts sensor outputs into actual part identifcation bits.  In 3 Sensor Mode, Inductive sees REJECT, Ultrasonic sees REJECT, SMALL, and ELECTRONIC, and Thru Beam sees ELECTRONIC AND LARGE.  In 4 Sensor Mode, Inductive sees REJECT, Ultrasonic sees REJECT, SMALL, and ELECTRONIC, Infrared Prox sees ELECTRONIC and LARGE, and Thru Beam sees only LARGE PART.

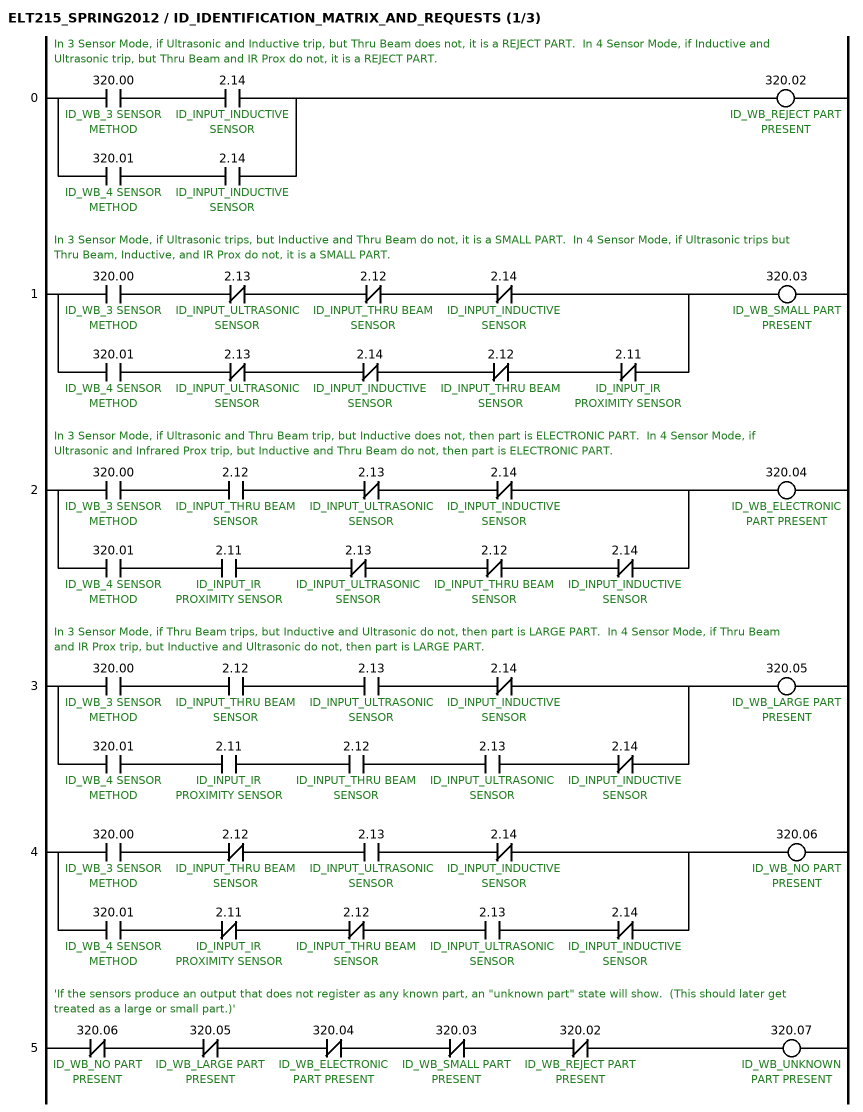
; rung 0: In 3 Sensor Mode, if Ultrasonic and Inductive trip, but Thru Beam does not, it is a REJECT PART.  In 4 Sensor Mode, if Inductive and Ultrasonic trip, but Thru Beam and IR Prox do not, it is a REJECT PART.
LD 320.00  ; ID_WB_3 SENSOR METHOD
AND 2.14  ; ID_INPUT_INDUCTIVE SENSOR
LD 320.01  ; ID_WB_4 SENSOR METHOD
AND 2.14  ; ID_INPUT_INDUCTIVE SENSOR
ORLD
OUT 320.02  ; ID_WB_REJECT PART PRESENT
; rung 1: In 3 Sensor Mode, if Ultrasonic trips, but Inductive and Thru Beam do not, it is a SMALL PART.  In 4 Sensor Mode, if Ultrasonic trips but Thru Beam, Inductive, and IR Prox do not, it is a SMALL PART.
LD 320.00  ; ID_WB_3 SENSOR METHOD
ANDNOT 2.13  ; ID_INPUT_ULTRASONIC SENSOR
ANDNOT 2.12  ; ID_INPUT_THRU BEAM SENSOR
ANDNOT 2.14  ; ID_INPUT_INDUCTIVE SENSOR
LD 320.01  ; ID_WB_4 SENSOR METHOD
ANDNOT 2.13  ; ID_INPUT_ULTRASONIC SENSOR
ANDNOT 2.14  ; ID_INPUT_INDUCTIVE SENSOR
ANDNOT 2.12  ; ID_INPUT_THRU BEAM SENSOR
ANDNOT 2.11  ; ID_INPUT_IR PROXIMITY SENSOR
ORLD
OUT 320.03  ; ID_WB_SMALL PART PRESENT
; rung 2: In 3 Sensor Mode, if Ultrasonic and Thru Beam trip, but Inductive does not, then part is ELECTRONIC PART.  In 4 Sensor Mode, if Ultrasonic and Infrared Prox trip, but Inductive and Thru Beam do not, then part is ELECTRONIC PART.
LD 320.00  ; ID_WB_3 SENSOR METHOD
AND 2.12  ; ID_INPUT_THRU BEAM SENSOR
ANDNOT 2.13  ; ID_INPUT_ULTRASONIC SENSOR
ANDNOT 2.14  ; ID_INPUT_INDUCTIVE SENSOR
LD 320.01  ; ID_WB_4 SENSOR METHOD
AND 2.11  ; ID_INPUT_IR PROXIMITY SENSOR
ANDNOT 2.13  ; ID_INPUT_ULTRASONIC SENSOR
ANDNOT 2.12  ; ID_INPUT_THRU BEAM SENSOR
ANDNOT 2.14  ; ID_INPUT_INDUCTIVE SENSOR
ORLD
OUT 320.04  ; ID_WB_ELECTRONIC PART PRESENT
; rung 3: In 3 Sensor Mode, if Thru Beam trips, but Inductive and Ultrasonic do not, then part is LARGE PART.  In 4 Sensor Mode, if Thru Beam and IR Prox trip, but Inductive and Ultrasonic do not, then part is LARGE PART.
LD 320.00  ; ID_WB_3 SENSOR METHOD
AND 2.12  ; ID_INPUT_THRU BEAM SENSOR
AND 2.13  ; ID_INPUT_ULTRASONIC SENSOR
ANDNOT 2.14  ; ID_INPUT_INDUCTIVE SENSOR
LD 320.01  ; ID_WB_4 SENSOR METHOD
AND 2.11  ; ID_INPUT_IR PROXIMITY SENSOR
AND 2.12  ; ID_INPUT_THRU BEAM SENSOR
AND 2.13  ; ID_INPUT_ULTRASONIC SENSOR
ANDNOT 2.14  ; ID_INPUT_INDUCTIVE SENSOR
ORLD
OUT 320.05  ; ID_WB_LARGE PART PRESENT
; rung 4
LD 320.00  ; ID_WB_3 SENSOR METHOD
ANDNOT 2.12  ; ID_INPUT_THRU BEAM SENSOR
AND 2.13  ; ID_INPUT_ULTRASONIC SENSOR
ANDNOT 2.14  ; ID_INPUT_INDUCTIVE SENSOR
LD 320.01  ; ID_WB_4 SENSOR METHOD
ANDNOT 2.11  ; ID_INPUT_IR PROXIMITY SENSOR
ANDNOT 2.12  ; ID_INPUT_THRU BEAM SENSOR
AND 2.13  ; ID_INPUT_ULTRASONIC SENSOR
ANDNOT 2.14  ; ID_INPUT_INDUCTIVE SENSOR
ORLD
OUT 320.06  ; ID_WB_NO PART PRESENT
; rung 5: 'If the sensors produce an output that does not register as any known part, an "unknown part" state will show.  (This should later get treated as a large or small part.)'
LDNOT 320.06  ; ID_WB_NO PART PRESENT
ANDNOT 320.05  ; ID_WB_LARGE PART PRESENT
ANDNOT 320.04  ; ID_WB_ELECTRONIC PART PRESENT
ANDNOT 320.03  ; ID_WB_SMALL PART PRESENT
ANDNOT 320.02  ; ID_WB_REJECT PART PRESENT
OUT 320.07  ; ID_WB_UNKNOWN PART PRESENT

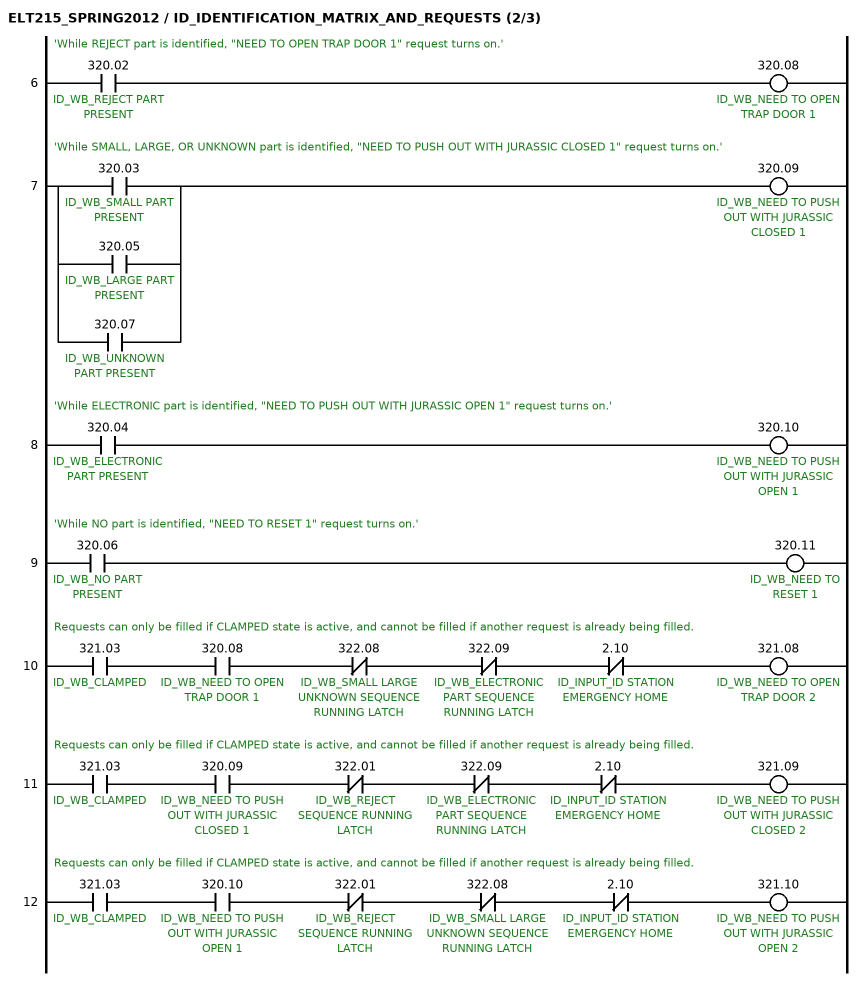
; rung 6: 'While REJECT part is identified, "NEED TO OPEN TRAP DOOR 1" request turns on.'
LD 320.02  ; ID_WB_REJECT PART PRESENT
OUT 320.08  ; ID_WB_NEED TO OPEN TRAP DOOR 1
; rung 7: 'While SMALL, LARGE, OR UNKNOWN part is identified, "NEED TO PUSH OUT WITH JURASSIC CLOSED 1" request turns on.'
LD 320.03  ; ID_WB_SMALL PART PRESENT
OR 320.05  ; ID_WB_LARGE PART PRESENT
OR 320.07  ; ID_WB_UNKNOWN PART PRESENT
OUT 320.09  ; ID_WB_NEED TO PUSH OUT WITH JURASSIC CLOSED 1
; rung 8: 'While ELECTRONIC part is identified, "NEED TO PUSH OUT WITH JURASSIC OPEN 1" request turns on.'
LD 320.04  ; ID_WB_ELECTRONIC PART PRESENT
OUT 320.10  ; ID_WB_NEED TO PUSH OUT WITH JURASSIC OPEN 1
; rung 9: 'While NO part is identified, "NEED TO RESET 1" request turns on.'
LD 320.06  ; ID_WB_NO PART PRESENT
OUT 320.11  ; ID_WB_NEED TO RESET 1
; rung 10: Requests can only be filled if CLAMPED state is active, and cannot be filled if another request is already being filled.
LD 321.03  ; ID_WB_CLAMPED
AND 320.08  ; ID_WB_NEED TO OPEN TRAP DOOR 1
ANDNOT 322.08  ; ID_WB_SMALL LARGE UNKNOWN SEQUENCE RUNNING LATCH
ANDNOT 322.09  ; ID_WB_ELECTRONIC PART SEQUENCE RUNNING LATCH
ANDNOT 2.10  ; ID_INPUT_ID STATION EMERGENCY HOME
OUT 321.08  ; ID_WB_NEED TO OPEN TRAP DOOR 2
; rung 11: Requests can only be filled if CLAMPED state is active, and cannot be filled if another request is already being filled.
LD 321.03  ; ID_WB_CLAMPED
AND 320.09  ; ID_WB_NEED TO PUSH OUT WITH JURASSIC CLOSED 1
ANDNOT 322.01  ; ID_WB_REJECT SEQUENCE RUNNING LATCH
ANDNOT 322.09  ; ID_WB_ELECTRONIC PART SEQUENCE RUNNING LATCH
ANDNOT 2.10  ; ID_INPUT_ID STATION EMERGENCY HOME
OUT 321.09  ; ID_WB_NEED TO PUSH OUT WITH JURASSIC CLOSED 2
; rung 12: Requests can only be filled if CLAMPED state is active, and cannot be filled if another request is already being filled.
LD 321.03  ; ID_WB_CLAMPED
AND 320.10  ; ID_WB_NEED TO PUSH OUT WITH JURASSIC OPEN 1
ANDNOT 322.01  ; ID_WB_REJECT SEQUENCE RUNNING LATCH
ANDNOT 322.08  ; ID_WB_SMALL LARGE UNKNOWN SEQUENCE RUNNING LATCH
ANDNOT 2.10  ; ID_INPUT_ID STATION EMERGENCY HOME
OUT 321.10  ; ID_WB_NEED TO PUSH OUT WITH JURASSIC OPEN 2

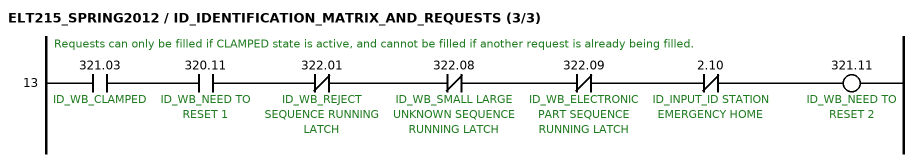
; rung 13: Requests can only be filled if CLAMPED state is active, and cannot be filled if another request is already being filled.
LD 321.03  ; ID_WB_CLAMPED
AND 320.11  ; ID_WB_NEED TO RESET 1
ANDNOT 322.01  ; ID_WB_REJECT SEQUENCE RUNNING LATCH
ANDNOT 322.08  ; ID_WB_SMALL LARGE UNKNOWN SEQUENCE RUNNING LATCH
ANDNOT 322.09  ; ID_WB_ELECTRONIC PART SEQUENCE RUNNING LATCH
ANDNOT 2.10  ; ID_INPUT_ID STATION EMERGENCY HOME
OUT 321.11  ; ID_WB_NEED TO RESET 2

### Section ID_OUTCOME_REJECT
; 'The actions required if a "REJECT" part is identified to be in the station.'

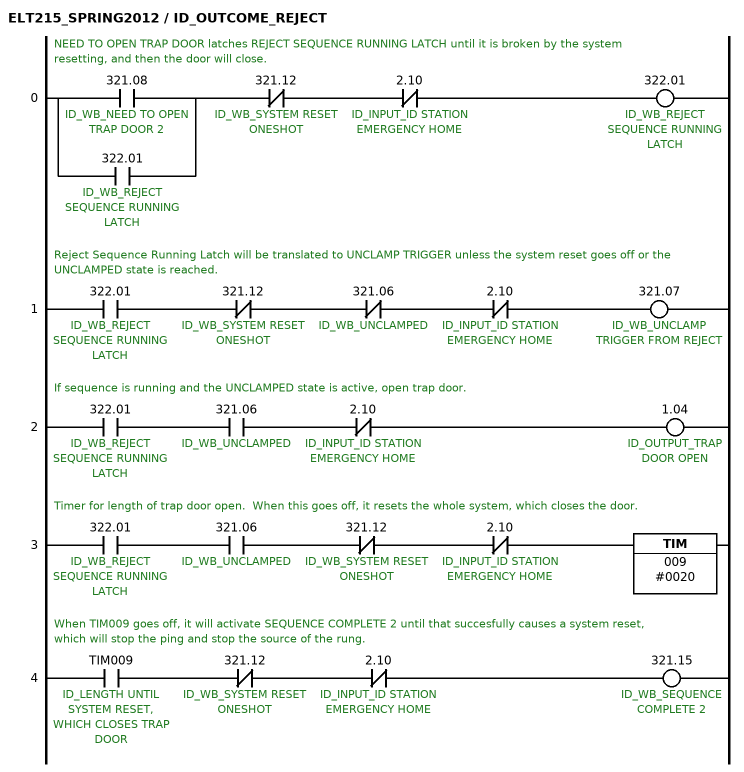
; rung 0: NEED TO OPEN TRAP DOOR latches REJECT SEQUENCE RUNNING LATCH until it is broken by the system resetting, and then the door will close.
LD 321.08  ; ID_WB_NEED TO OPEN TRAP DOOR 2
OR 322.01  ; ID_WB_REJECT SEQUENCE RUNNING LATCH
ANDNOT 321.12  ; ID_WB_SYSTEM RESET ONESHOT
ANDNOT 2.10  ; ID_INPUT_ID STATION EMERGENCY HOME
OUT 322.01  ; ID_WB_REJECT SEQUENCE RUNNING LATCH
; rung 1: Reject Sequence Running Latch will be translated to UNCLAMP TRIGGER unless the system reset goes off or the UNCLAMPED state is reached.
LD 322.01  ; ID_WB_REJECT SEQUENCE RUNNING LATCH
ANDNOT 321.12  ; ID_WB_SYSTEM RESET ONESHOT
ANDNOT 321.06  ; ID_WB_UNCLAMPED
ANDNOT 2.10  ; ID_INPUT_ID STATION EMERGENCY HOME
OUT 321.07  ; ID_WB_UNCLAMP TRIGGER FROM REJECT
; rung 2: If sequence is running and the UNCLAMPED state is active, open trap door.
LD 322.01  ; ID_WB_REJECT SEQUENCE RUNNING LATCH
AND 321.06  ; ID_WB_UNCLAMPED
ANDNOT 2.10  ; ID_INPUT_ID STATION EMERGENCY HOME
OUT 1.04  ; ID_OUTPUT_TRAP DOOR OPEN
; rung 3: Timer for length of trap door open.  When this goes off, it resets the whole system, which closes the door.
LD 322.01  ; ID_WB_REJECT SEQUENCE RUNNING LATCH
AND 321.06  ; ID_WB_UNCLAMPED
ANDNOT 321.12  ; ID_WB_SYSTEM RESET ONESHOT
ANDNOT 2.10  ; ID_INPUT_ID STATION EMERGENCY HOME
TIM 009 #0020
; rung 4: When TIM009 goes off, it will activate SEQUENCE COMPLETE 2 until that succesfully causes a system reset, which will stop the ping and stop the source of the rung.
LD TIM009  ; ID_LENGTH UNTIL SYSTEM RESET, WHICH CLOSES TRAP DOOR
ANDNOT 321.12  ; ID_WB_SYSTEM RESET ONESHOT
ANDNOT 2.10  ; ID_INPUT_ID STATION EMERGENCY HOME
OUT 321.15  ; ID_WB_SEQUENCE COMPLETE 2

### Section ID_OUTCOME_SMALL_LARGE_UNKNOWN
; The actions required if the part identified in the station is SMALL, LARGE, or UNKNOWN.  (They all have the same outcome.)  This triggers the same push sequence as the ELECTRONIC PART except it does not raise the JURASSIC GATE or wait for the JURASSIC GATE to open.

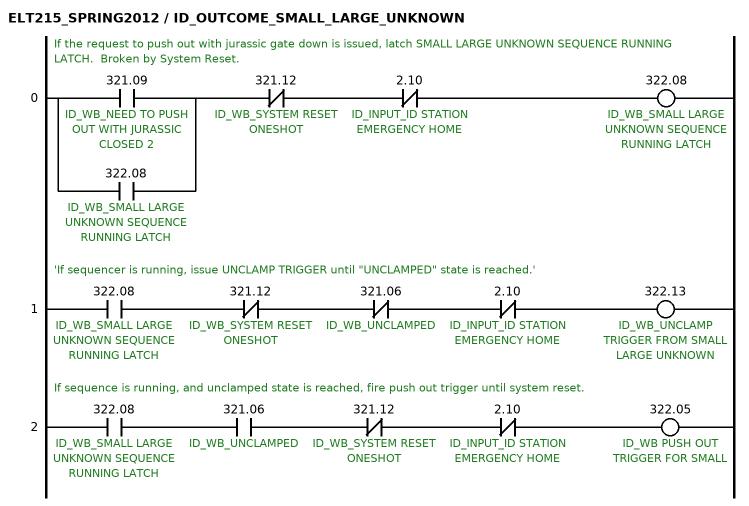
; rung 0: If the request to push out with jurassic gate down is issued, latch SMALL LARGE UNKNOWN SEQUENCE RUNNING LATCH.  Broken by System Reset.
LD 321.09  ; ID_WB_NEED TO PUSH OUT WITH JURASSIC CLOSED 2
OR 322.08  ; ID_WB_SMALL LARGE UNKNOWN SEQUENCE RUNNING LATCH
ANDNOT 321.12  ; ID_WB_SYSTEM RESET ONESHOT
ANDNOT 2.10  ; ID_INPUT_ID STATION EMERGENCY HOME
OUT 322.08  ; ID_WB_SMALL LARGE UNKNOWN SEQUENCE RUNNING LATCH
; rung 1: 'If sequencer is running, issue UNCLAMP TRIGGER until "UNCLAMPED" state is reached.'
LD 322.08  ; ID_WB_SMALL LARGE UNKNOWN SEQUENCE RUNNING LATCH
ANDNOT 321.12  ; ID_WB_SYSTEM RESET ONESHOT
ANDNOT 321.06  ; ID_WB_UNCLAMPED
ANDNOT 2.10  ; ID_INPUT_ID STATION EMERGENCY HOME
OUT 322.13  ; ID_WB_UNCLAMP TRIGGER FROM SMALL LARGE UNKNOWN
; rung 2: If sequence is running, and unclamped state is reached, fire push out trigger until system reset.
LD 322.08  ; ID_WB_SMALL LARGE UNKNOWN SEQUENCE RUNNING LATCH
AND 321.06  ; ID_WB_UNCLAMPED
ANDNOT 321.12  ; ID_WB_SYSTEM RESET ONESHOT
ANDNOT 2.10  ; ID_INPUT_ID STATION EMERGENCY HOME
OUT 322.05  ; ID_WB PUSH OUT TRIGGER FOR SMALL

### Section ID_OUTCOME_ELECTRONIC
; The actions required if the part identified to be in the station is an ELECTRONIC PART.  This triggers the same PUSH sequence as the SMALL/LARGE/UNKNOWN PART, but waits for the JURASSIC GATE to open.

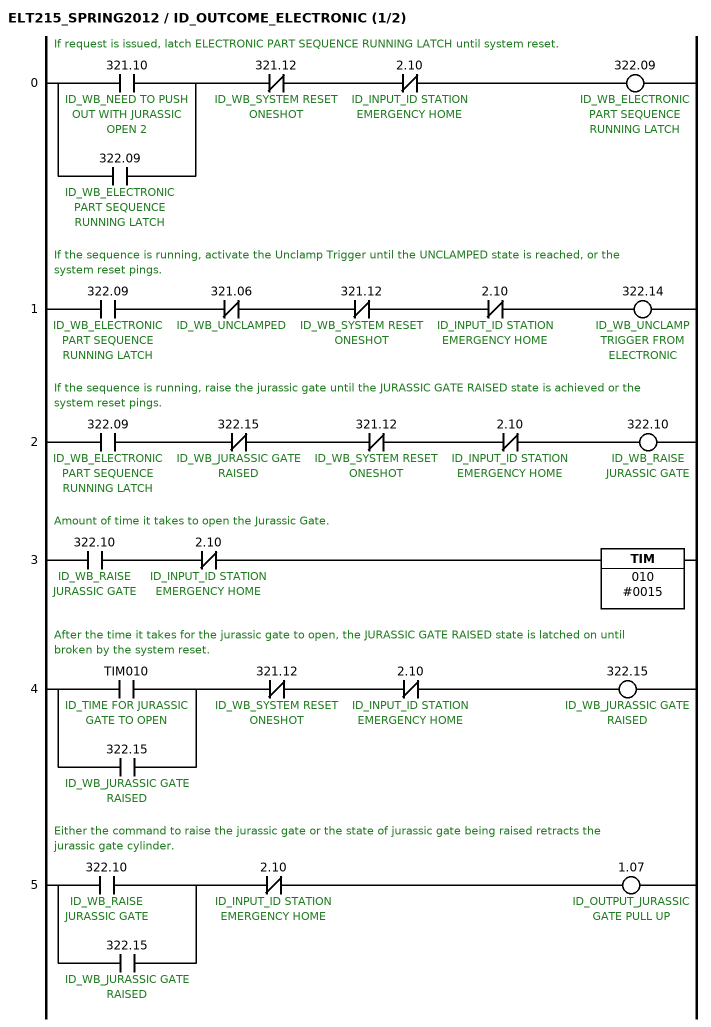
; rung 0: If request is issued, latch ELECTRONIC PART SEQUENCE RUNNING LATCH until system reset.
LD 321.10  ; ID_WB_NEED TO PUSH OUT WITH JURASSIC OPEN 2
OR 322.09  ; ID_WB_ELECTRONIC PART SEQUENCE RUNNING LATCH
ANDNOT 321.12  ; ID_WB_SYSTEM RESET ONESHOT
ANDNOT 2.10  ; ID_INPUT_ID STATION EMERGENCY HOME
OUT 322.09  ; ID_WB_ELECTRONIC PART SEQUENCE RUNNING LATCH
; rung 1: If the sequence is running, activate the Unclamp Trigger until the UNCLAMPED state is reached, or the system reset pings.
LD 322.09  ; ID_WB_ELECTRONIC PART SEQUENCE RUNNING LATCH
ANDNOT 321.06  ; ID_WB_UNCLAMPED
ANDNOT 321.12  ; ID_WB_SYSTEM RESET ONESHOT
ANDNOT 2.10  ; ID_INPUT_ID STATION EMERGENCY HOME
OUT 322.14  ; ID_WB_UNCLAMP TRIGGER FROM ELECTRONIC
; rung 2: If the sequence is running, raise the jurassic gate until the JURASSIC GATE RAISED state is achieved or the system reset pings.
LD 322.09  ; ID_WB_ELECTRONIC PART SEQUENCE RUNNING LATCH
ANDNOT 322.15  ; ID_WB_JURASSIC GATE RAISED
ANDNOT 321.12  ; ID_WB_SYSTEM RESET ONESHOT
ANDNOT 2.10  ; ID_INPUT_ID STATION EMERGENCY HOME
OUT 322.10  ; ID_WB_RAISE JURASSIC GATE
; rung 3: Amount of time it takes to open the Jurassic Gate.
LD 322.10  ; ID_WB_RAISE JURASSIC GATE
ANDNOT 2.10  ; ID_INPUT_ID STATION EMERGENCY HOME
TIM 010 #0015
; rung 4: After the time it takes for the jurassic gate to open, the JURASSIC GATE RAISED state is latched on until broken by the system reset.
LD TIM010  ; ID_TIME FOR JURASSIC GATE TO OPEN
OR 322.15  ; ID_WB_JURASSIC GATE RAISED
ANDNOT 321.12  ; ID_WB_SYSTEM RESET ONESHOT
ANDNOT 2.10  ; ID_INPUT_ID STATION EMERGENCY HOME
OUT 322.15  ; ID_WB_JURASSIC GATE RAISED
; rung 5: Either the command to raise the jurassic gate or the state of jurassic gate being raised retracts the jurassic gate cylinder.
LD 322.10  ; ID_WB_RAISE JURASSIC GATE
OR 322.15  ; ID_WB_JURASSIC GATE RAISED
ANDNOT 2.10  ; ID_INPUT_ID STATION EMERGENCY HOME
OUT 1.07  ; ID_OUTPUT_JURASSIC GATE PULL UP

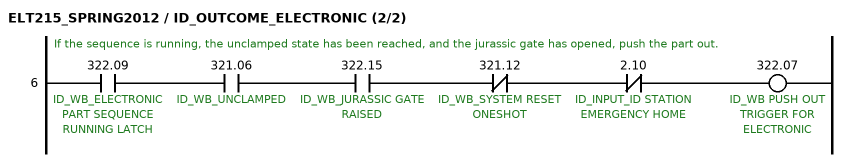
; rung 6: If the sequence is running, the unclamped state has been reached, and the jurassic gate has opened, push the part out.
LD 322.09  ; ID_WB_ELECTRONIC PART SEQUENCE RUNNING LATCH
AND 321.06  ; ID_WB_UNCLAMPED
AND 322.15  ; ID_WB_JURASSIC GATE RAISED
ANDNOT 321.12  ; ID_WB_SYSTEM RESET ONESHOT
ANDNOT 2.10  ; ID_INPUT_ID STATION EMERGENCY HOME
OUT 322.07  ; ID_WB PUSH OUT TRIGGER FOR ELECTRONIC

### Section ID_PUSH_CONCLUSION
; Contains the pushing out sequence of actions from the result of either SMALL, LARGE, UNKNOWN, or ELECTRONIC parts.

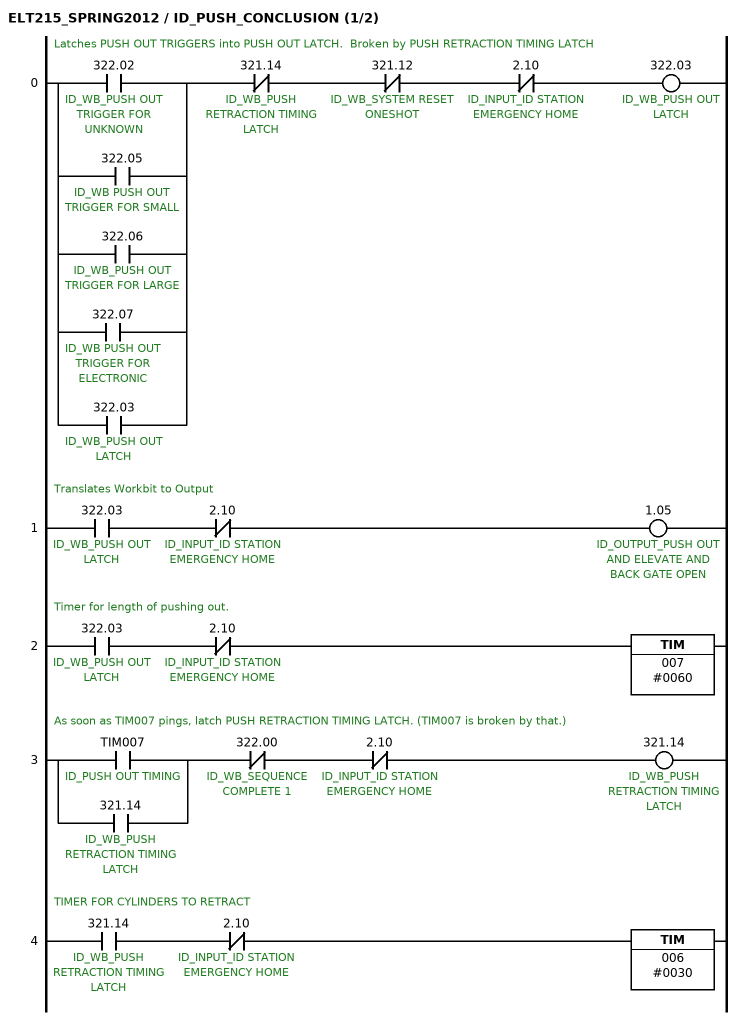
; rung 0: Latches PUSH OUT TRIGGERS into PUSH OUT LATCH.  Broken by PUSH RETRACTION TIMING LATCH
LD 322.02  ; ID_WB_PUSH OUT TRIGGER FOR UNKNOWN
OR 322.05  ; ID_WB PUSH OUT TRIGGER FOR SMALL
OR 322.06  ; ID_WB_PUSH OUT TRIGGER FOR LARGE
OR 322.07  ; ID_WB PUSH OUT TRIGGER FOR ELECTRONIC
OR 322.03  ; ID_WB_PUSH OUT LATCH
ANDNOT 321.14  ; ID_WB_PUSH RETRACTION TIMING LATCH
ANDNOT 321.12  ; ID_WB_SYSTEM RESET ONESHOT
ANDNOT 2.10  ; ID_INPUT_ID STATION EMERGENCY HOME
OUT 322.03  ; ID_WB_PUSH OUT LATCH
; rung 1: Translates Workbit to Output
LD 322.03  ; ID_WB_PUSH OUT LATCH
ANDNOT 2.10  ; ID_INPUT_ID STATION EMERGENCY HOME
OUT 1.05  ; ID_OUTPUT_PUSH OUT AND ELEVATE AND BACK GATE OPEN
; rung 2: Timer for length of pushing out.
LD 322.03  ; ID_WB_PUSH OUT LATCH
ANDNOT 2.10  ; ID_INPUT_ID STATION EMERGENCY HOME
TIM 007 #0060
; rung 3: As soon as TIM007 pings, latch PUSH RETRACTION TIMING LATCH. (TIM007 is broken by that.)
LD TIM007  ; ID_PUSH OUT TIMING
OR 321.14  ; ID_WB_PUSH RETRACTION TIMING LATCH
ANDNOT 322.00  ; ID_WB_SEQUENCE COMPLETE 1
ANDNOT 2.10  ; ID_INPUT_ID STATION EMERGENCY HOME
OUT 321.14  ; ID_WB_PUSH RETRACTION TIMING LATCH
; rung 4: TIMER FOR CYLINDERS TO RETRACT
LD 321.14  ; ID_WB_PUSH RETRACTION TIMING LATCH
ANDNOT 2.10  ; ID_INPUT_ID STATION EMERGENCY HOME
TIM 006 #0030

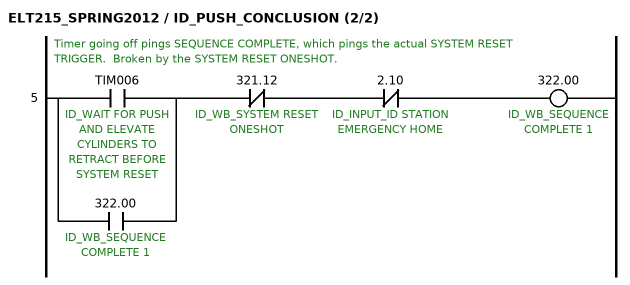
; rung 5: Timer going off pings SEQUENCE COMPLETE, which pings the actual SYSTEM RESET TRIGGER.  Broken by the SYSTEM RESET ONESHOT.
LD TIM006  ; ID_WAIT FOR PUSH AND ELEVATE CYLINDERS TO RETRACT BEFORE SYSTEM RESET
OR 322.00  ; ID_WB_SEQUENCE COMPLETE 1
ANDNOT 321.12  ; ID_WB_SYSTEM RESET ONESHOT
ANDNOT 2.10  ; ID_INPUT_ID STATION EMERGENCY HOME
OUT 322.00  ; ID_WB_SEQUENCE COMPLETE 1

### Section ID_SYSTEM_RESET_ONESHOT
; Either from no part or from sequence complete, the ladder logic for system resets.

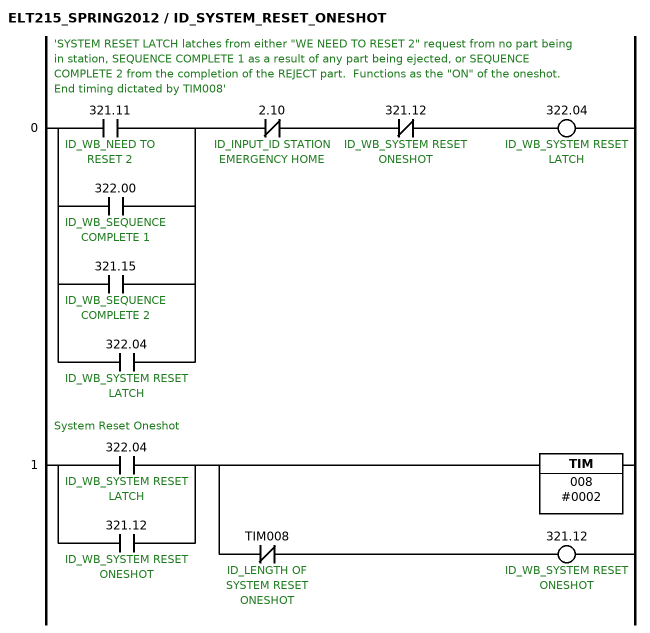
; rung 0: 'SYSTEM RESET LATCH latches from either "WE NEED TO RESET 2" request from no part being in station, SEQUENCE COMPLETE 1 as a result of any part being ejected, or SEQUENCE COMPLETE 2 from the completion of the REJECT part.  Functions as the "ON" of the oneshot.  End timing dictated by TIM008'
LD 321.11  ; ID_WB_NEED TO RESET 2
OR 322.00  ; ID_WB_SEQUENCE COMPLETE 1
OR 321.15  ; ID_WB_SEQUENCE COMPLETE 2
OR 322.04  ; ID_WB_SYSTEM RESET LATCH
ANDNOT 2.10  ; ID_INPUT_ID STATION EMERGENCY HOME
ANDNOT 321.12  ; ID_WB_SYSTEM RESET ONESHOT
OUT 322.04  ; ID_WB_SYSTEM RESET LATCH
; rung 1: System Reset Oneshot
LD 322.04  ; ID_WB_SYSTEM RESET LATCH
OR 321.12  ; ID_WB_SYSTEM RESET ONESHOT
TIM 008 #0002
ANDNOT TIM008  ; ID_LENGTH OF SYSTEM RESET ONESHOT
OUT 321.12  ; ID_WB_SYSTEM RESET ONESHOT

### Section ID_OBSERVATION_ONLY

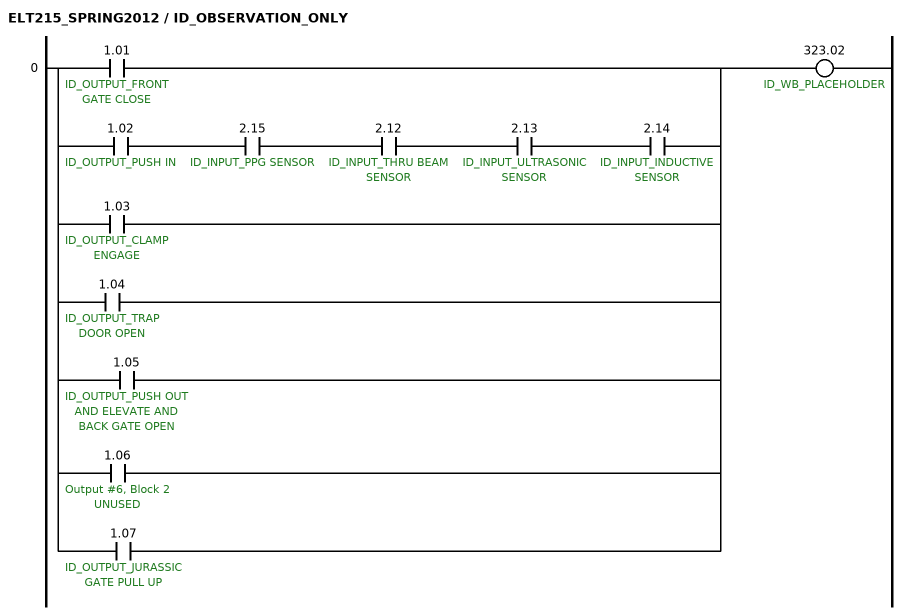
; rung 0
LD 1.01  ; ID_OUTPUT_FRONT GATE CLOSE
LD 1.02  ; ID_OUTPUT_PUSH IN
AND 2.15  ; ID_INPUT_PPG SENSOR
AND 2.12  ; ID_INPUT_THRU BEAM SENSOR
AND 2.13  ; ID_INPUT_ULTRASONIC SENSOR
AND 2.14  ; ID_INPUT_INDUCTIVE SENSOR
ORLD
LD 1.03  ; ID_OUTPUT_CLAMP ENGAGE
OR 1.04  ; ID_OUTPUT_TRAP DOOR OPEN
OR 1.05  ; ID_OUTPUT_PUSH OUT AND ELEVATE AND BACK GATE OPEN
OR 1.06  ; Output #6, Block 2 UNUSED
OR 1.07  ; ID_OUTPUT_JURASSIC GATE PULL UP
ORLD
OUT 323.02  ; ID_WB_PLACEHOLDER

### Section T_GETTING_PART_RESEATING_AND_LOCKING
; Ladder logic that gets the part into the testing station.

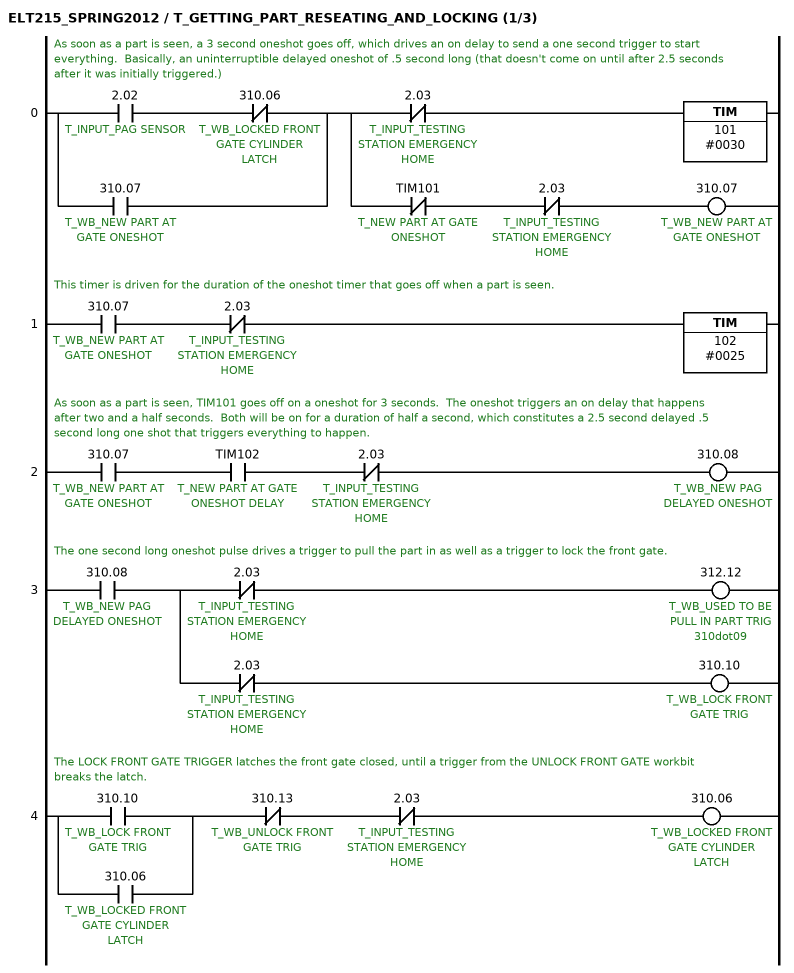
; rung 0: As soon as a part is seen, a 3 second oneshot goes off, which drives an on delay to send a one second trigger to start everything.  Basically, an uninterruptible delayed oneshot of .5 second long (that doesn't come on until after 2.5 seconds after it was initially triggered.)
LD 2.02  ; T_INPUT_PAG SENSOR
ANDNOT 310.06  ; T_WB_LOCKED FRONT GATE CYLINDER LATCH
OR 310.07  ; T_WB_NEW PART AT GATE ONESHOT
OUT TR0
ANDNOT 2.03  ; T_INPUT_TESTING STATION EMERGENCY HOME
TIM 101 #0030
LD TR0
ANDNOT TIM101  ; T_NEW PART AT GATE ONESHOT
ANDNOT 2.03  ; T_INPUT_TESTING STATION EMERGENCY HOME
OUT 310.07  ; T_WB_NEW PART AT GATE ONESHOT
; rung 1: This timer is driven for the duration of the oneshot timer that goes off when a part is seen.
LD 310.07  ; T_WB_NEW PART AT GATE ONESHOT
ANDNOT 2.03  ; T_INPUT_TESTING STATION EMERGENCY HOME
TIM 102 #0025
; rung 2: As soon as a part is seen, TIM101 goes off on a oneshot for 3 seconds.  The oneshot triggers an on delay that happens after two and a half seconds.  Both will be on for a duration of half a second, which constitutes a 2.5 second delayed .5 second long one shot that triggers everything to happen.
LD 310.07  ; T_WB_NEW PART AT GATE ONESHOT
AND TIM102  ; T_NEW PART AT GATE ONESHOT DELAY
ANDNOT 2.03  ; T_INPUT_TESTING STATION EMERGENCY HOME
OUT 310.08  ; T_WB_NEW PAG DELAYED ONESHOT
; rung 3: The one second long oneshot pulse drives a trigger to pull the part in as well as a trigger to lock the front gate.
LD 310.08  ; T_WB_NEW PAG DELAYED ONESHOT
OUT TR0
ANDNOT 2.03  ; T_INPUT_TESTING STATION EMERGENCY HOME
OUT 312.12  ; T_WB_USED TO BE PULL IN PART TRIG 310dot09
LD TR0
ANDNOT 2.03  ; T_INPUT_TESTING STATION EMERGENCY HOME
OUT 310.10  ; T_WB_LOCK FRONT GATE TRIG
; rung 4: The LOCK FRONT GATE TRIGGER latches the front gate closed, until a trigger from the UNLOCK FRONT GATE workbit breaks the latch.
LD 310.10  ; T_WB_LOCK FRONT GATE TRIG
OR 310.06  ; T_WB_LOCKED FRONT GATE CYLINDER LATCH
ANDNOT 310.13  ; T_WB_UNLOCK FRONT GATE TRIG
ANDNOT 2.03  ; T_INPUT_TESTING STATION EMERGENCY HOME
OUT 310.06  ; T_WB_LOCKED FRONT GATE CYLINDER LATCH

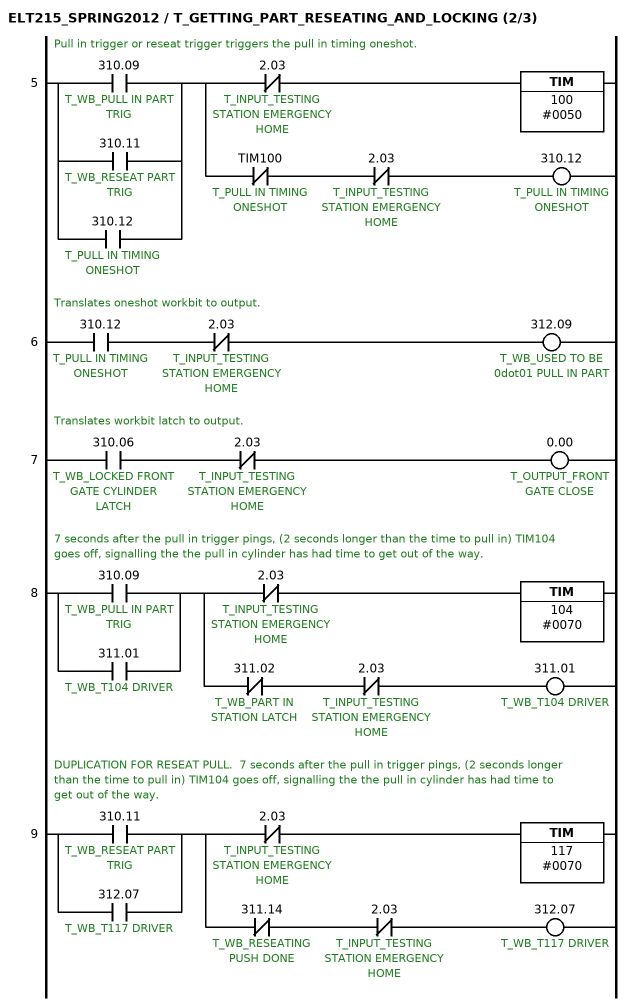
; rung 5: Pull in trigger or reseat trigger triggers the pull in timing oneshot.
LD 310.09  ; T_WB_PULL IN PART TRIG
OR 310.11  ; T_WB_RESEAT PART TRIG
OR 310.12  ; T_PULL IN TIMING ONESHOT
OUT TR0
ANDNOT 2.03  ; T_INPUT_TESTING STATION EMERGENCY HOME
TIM 100 #0050
LD TR0
ANDNOT TIM100  ; T_PULL IN TIMING ONESHOT
ANDNOT 2.03  ; T_INPUT_TESTING STATION EMERGENCY HOME
OUT 310.12  ; T_PULL IN TIMING ONESHOT
; rung 6: Translates oneshot workbit to output.
LD 310.12  ; T_PULL IN TIMING ONESHOT
ANDNOT 2.03  ; T_INPUT_TESTING STATION EMERGENCY HOME
OUT 312.09  ; T_WB_USED TO BE 0dot01 PULL IN PART
; rung 7: Translates workbit latch to output.
LD 310.06  ; T_WB_LOCKED FRONT GATE CYLINDER LATCH
ANDNOT 2.03  ; T_INPUT_TESTING STATION EMERGENCY HOME
OUT 0.00  ; T_OUTPUT_FRONT GATE CLOSE
; rung 8: 7 seconds after the pull in trigger pings, (2 seconds longer than the time to pull in) TIM104 goes off, signalling the the pull in cylinder has had time to get out of the way.
LD 310.09  ; T_WB_PULL IN PART TRIG
OR 311.01  ; T_WB_T104 DRIVER
OUT TR0
ANDNOT 2.03  ; T_INPUT_TESTING STATION EMERGENCY HOME
TIM 104 #0070
LD TR0
ANDNOT 311.02  ; T_WB_PART IN STATION LATCH
ANDNOT 2.03  ; T_INPUT_TESTING STATION EMERGENCY HOME
OUT 311.01  ; T_WB_T104 DRIVER
; rung 9: DUPLICATION FOR RESEAT PULL.  7 seconds after the pull in trigger pings, (2 seconds longer than the time to pull in) TIM104 goes off, signalling the the pull in cylinder has had time to get out of the way.
LD 310.11  ; T_WB_RESEAT PART TRIG
OR 312.07  ; T_WB_T117 DRIVER
OUT TR0
ANDNOT 2.03  ; T_INPUT_TESTING STATION EMERGENCY HOME
TIM 117 #0070
LD TR0
ANDNOT 311.14  ; T_WB_RESEATING PUSH DONE
ANDNOT 2.03  ; T_INPUT_TESTING STATION EMERGENCY HOME
OUT 312.07  ; T_WB_T117 DRIVER

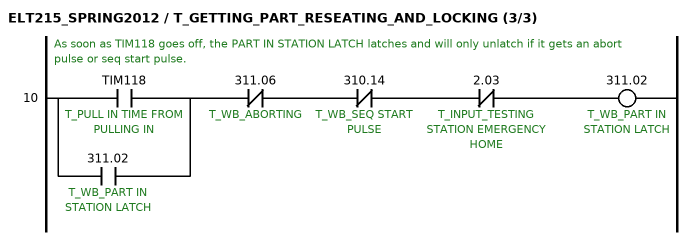
; rung 10: As soon as TIM118 goes off, the PART IN STATION LATCH latches and will only unlatch if it gets an abort pulse or seq start pulse.
LD TIM118  ; T_PULL IN TIME FROM PULLING IN
OR 311.02  ; T_WB_PART IN STATION LATCH
ANDNOT 311.06  ; T_WB_ABORTING
ANDNOT 310.14  ; T_WB_SEQ START PULSE
ANDNOT 2.03  ; T_INPUT_TESTING STATION EMERGENCY HOME
OUT 311.02  ; T_WB_PART IN STATION LATCH

### Section T_NEW_PULL_IN_BEHAVIOR

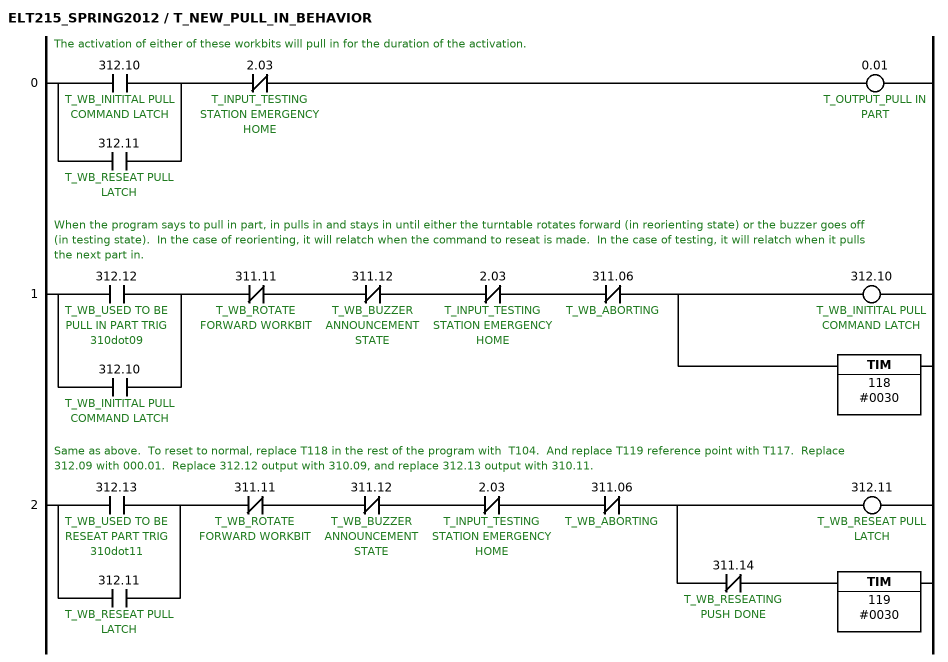
; rung 0: The activation of either of these workbits will pull in for the duration of the activation.
LD 312.10  ; T_WB_INITITAL PULL COMMAND LATCH
OR 312.11  ; T_WB_RESEAT PULL LATCH
ANDNOT 2.03  ; T_INPUT_TESTING STATION EMERGENCY HOME
OUT 0.01  ; T_OUTPUT_PULL IN PART
; rung 1: When the program says to pull in part, in pulls in and stays in until either the turntable rotates forward (in reorienting state) or the buzzer goes off (in testing state).  In the case of reorienting, it will relatch when the command to reseat is made.  In the case of testing, it will relatch when it pulls the next part in.
LD 312.12  ; T_WB_USED TO BE PULL IN PART TRIG 310dot09
OR 312.10  ; T_WB_INITITAL PULL COMMAND LATCH
ANDNOT 311.11  ; T_WB_ROTATE FORWARD WORKBIT
ANDNOT 311.12  ; T_WB_BUZZER ANNOUNCEMENT STATE
ANDNOT 2.03  ; T_INPUT_TESTING STATION EMERGENCY HOME
ANDNOT 311.06  ; T_WB_ABORTING
OUT 312.10  ; T_WB_INITITAL PULL COMMAND LATCH
TIM 118 #0030
; rung 2: Same as above.  To reset to normal, replace T118 in the rest of the program with  T104.  And replace T119 reference point with T117.  Replace 312.09 with 000.01.  Replace 312.12 output with 310.09, and replace 312.13 output with 310.11.
LD 312.13  ; T_WB_USED TO BE RESEAT PART TRIG 310dot11
OR 312.11  ; T_WB_RESEAT PULL LATCH
ANDNOT 311.11  ; T_WB_ROTATE FORWARD WORKBIT
ANDNOT 311.12  ; T_WB_BUZZER ANNOUNCEMENT STATE
ANDNOT 2.03  ; T_INPUT_TESTING STATION EMERGENCY HOME
ANDNOT 311.06  ; T_WB_ABORTING
OUT 312.11  ; T_WB_RESEAT PULL LATCH
ANDNOT 311.14  ; T_WB_RESEATING PUSH DONE
TIM 119 #0030

### Section T_CLAMPED_STATE
; 'Sets the "CLAMPED" state and manages UNCLAMP interrupts to that.'

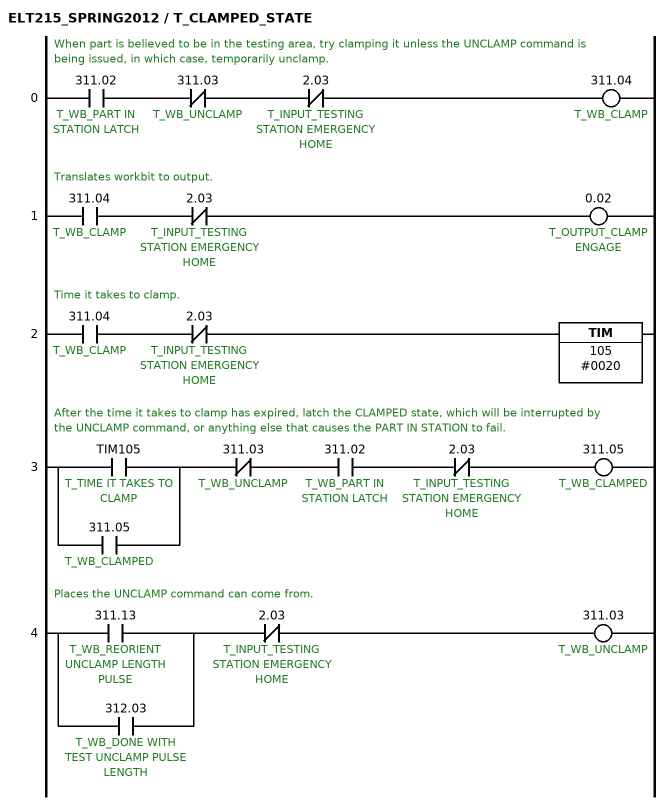
; rung 0: When part is believed to be in the testing area, try clamping it unless the UNCLAMP command is being issued, in which case, temporarily unclamp.
LD 311.02  ; T_WB_PART IN STATION LATCH
ANDNOT 311.03  ; T_WB_UNCLAMP
ANDNOT 2.03  ; T_INPUT_TESTING STATION EMERGENCY HOME
OUT 311.04  ; T_WB_CLAMP
; rung 1: Translates workbit to output.
LD 311.04  ; T_WB_CLAMP
ANDNOT 2.03  ; T_INPUT_TESTING STATION EMERGENCY HOME
OUT 0.02  ; T_OUTPUT_CLAMP ENGAGE
; rung 2: Time it takes to clamp.
LD 311.04  ; T_WB_CLAMP
ANDNOT 2.03  ; T_INPUT_TESTING STATION EMERGENCY HOME
TIM 105 #0020
; rung 3: After the time it takes to clamp has expired, latch the CLAMPED state, which will be interrupted by the UNCLAMP command, or anything else that causes the PART IN STATION to fail.
LD TIM105  ; T_TIME IT TAKES TO CLAMP
OR 311.05  ; T_WB_CLAMPED
ANDNOT 311.03  ; T_WB_UNCLAMP
AND 311.02  ; T_WB_PART IN STATION LATCH
ANDNOT 2.03  ; T_INPUT_TESTING STATION EMERGENCY HOME
OUT 311.05  ; T_WB_CLAMPED
; rung 4: Places the UNCLAMP command can come from.
LD 311.13  ; T_WB_REORIENT UNCLAMP LENGTH PULSE
OR 312.03  ; T_WB_DONE WITH TEST UNCLAMP PULSE LENGTH
ANDNOT 2.03  ; T_INPUT_TESTING STATION EMERGENCY HOME
OUT 311.03  ; T_WB_UNCLAMP

### Section T_ORIENTATION_STATES_AND_REQUESTS
; Combinational logic that converts sensor outputs into orientation identifcation work bits and then into action requests.

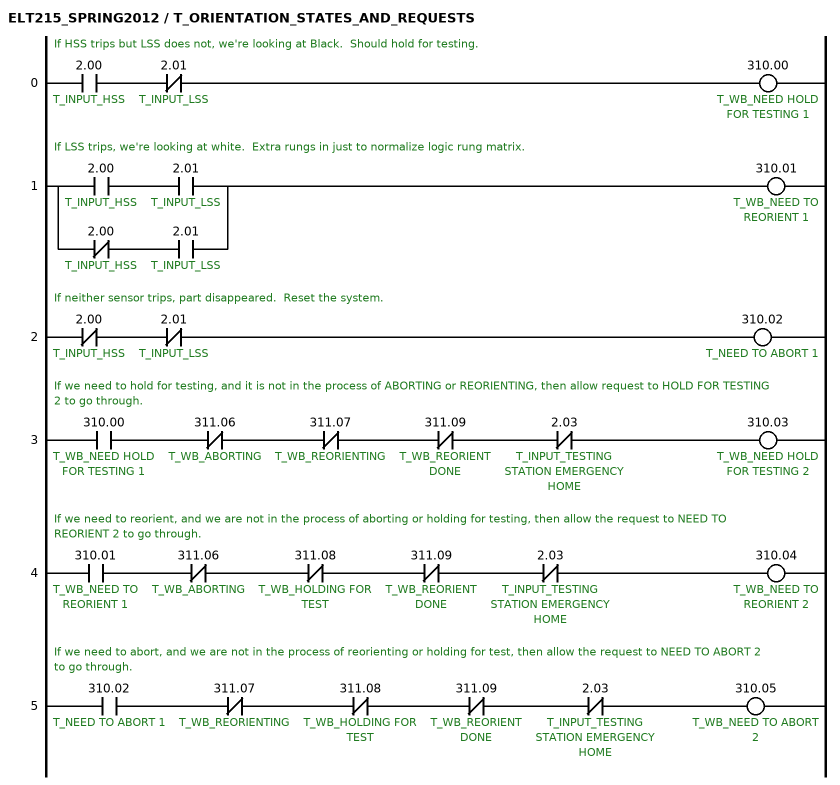
; rung 0: If HSS trips but LSS does not, we're looking at Black.  Should hold for testing.
LD 2.00  ; T_INPUT_HSS
ANDNOT 2.01  ; T_INPUT_LSS
OUT 310.00  ; T_WB_NEED HOLD FOR TESTING 1
; rung 1: If LSS trips, we're looking at white.  Extra rungs in just to normalize logic rung matrix.
LD 2.00  ; T_INPUT_HSS
AND 2.01  ; T_INPUT_LSS
LDNOT 2.00  ; T_INPUT_HSS
AND 2.01  ; T_INPUT_LSS
ORLD
OUT 310.01  ; T_WB_NEED TO REORIENT 1
; rung 2: If neither sensor trips, part disappeared.  Reset the system.
LDNOT 2.00  ; T_INPUT_HSS
ANDNOT 2.01  ; T_INPUT_LSS
OUT 310.02  ; T_NEED TO ABORT 1
; rung 3: If we need to hold for testing, and it is not in the process of ABORTING or REORIENTING, then allow request to HOLD FOR TESTING 2 to go through.
LD 310.00  ; T_WB_NEED HOLD FOR TESTING 1
ANDNOT 311.06  ; T_WB_ABORTING
ANDNOT 311.07  ; T_WB_REORIENTING
ANDNOT 311.09  ; T_WB_REORIENT DONE
ANDNOT 2.03  ; T_INPUT_TESTING STATION EMERGENCY HOME
OUT 310.03  ; T_WB_NEED HOLD FOR TESTING 2
; rung 4: If we need to reorient, and we are not in the process of aborting or holding for testing, then allow the request to NEED TO REORIENT 2 to go through.
LD 310.01  ; T_WB_NEED TO REORIENT 1
ANDNOT 311.06  ; T_WB_ABORTING
ANDNOT 311.08  ; T_WB_HOLDING FOR TEST
ANDNOT 311.09  ; T_WB_REORIENT DONE
ANDNOT 2.03  ; T_INPUT_TESTING STATION EMERGENCY HOME
OUT 310.04  ; T_WB_NEED TO REORIENT 2
; rung 5: If we need to abort, and we are not in the process of reorienting or holding for test, then allow the request to NEED TO ABORT 2 to go through.
LD 310.02  ; T_NEED TO ABORT 1
ANDNOT 311.07  ; T_WB_REORIENTING
ANDNOT 311.08  ; T_WB_HOLDING FOR TEST
ANDNOT 311.09  ; T_WB_REORIENT DONE
ANDNOT 2.03  ; T_INPUT_TESTING STATION EMERGENCY HOME
OUT 310.05  ; T_WB_NEED TO ABORT 2

### Section T_REORIENTING
; Ladder logic that performs the actions necessary to accept a second tier request to reorient the part and physically reorient the part itself by 90 degrees.

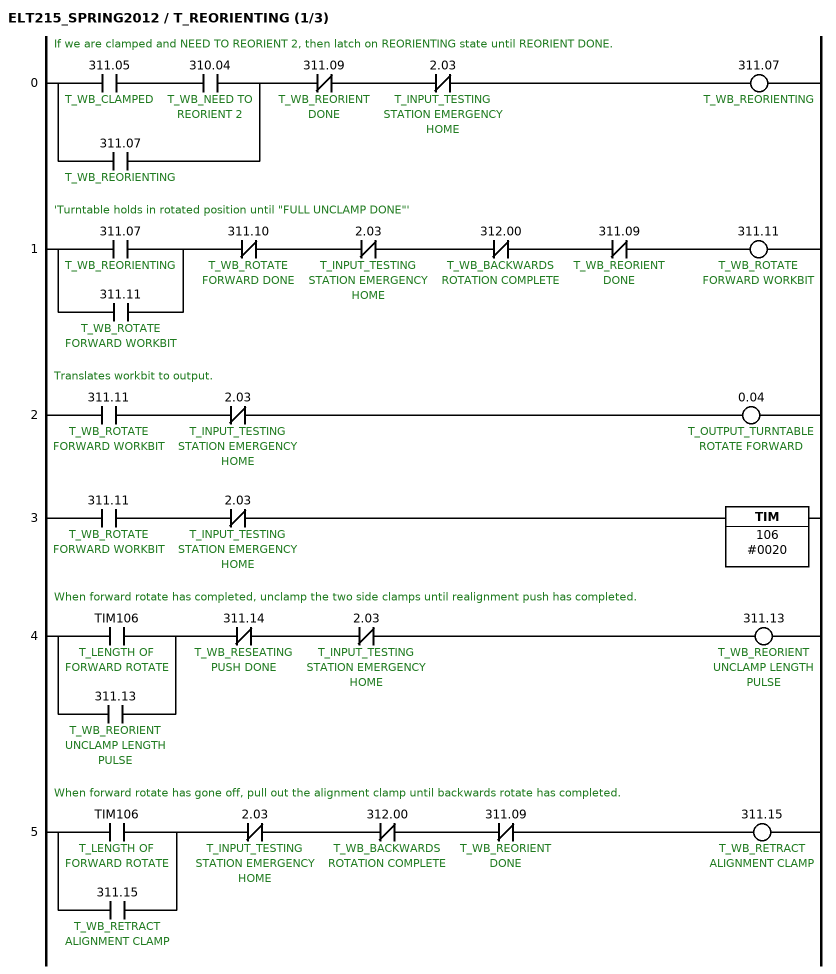
; rung 0: If we are clamped and NEED TO REORIENT 2, then latch on REORIENTING state until REORIENT DONE.
LD 311.05  ; T_WB_CLAMPED
AND 310.04  ; T_WB_NEED TO REORIENT 2
OR 311.07  ; T_WB_REORIENTING
ANDNOT 311.09  ; T_WB_REORIENT DONE
ANDNOT 2.03  ; T_INPUT_TESTING STATION EMERGENCY HOME
OUT 311.07  ; T_WB_REORIENTING
; rung 1: 'Turntable holds in rotated position until "FULL UNCLAMP DONE"'
LD 311.07  ; T_WB_REORIENTING
OR 311.11  ; T_WB_ROTATE FORWARD WORKBIT
ANDNOT 311.10  ; T_WB_ROTATE FORWARD DONE
ANDNOT 2.03  ; T_INPUT_TESTING STATION EMERGENCY HOME
ANDNOT 312.00  ; T_WB_BACKWARDS ROTATION COMPLETE
ANDNOT 311.09  ; T_WB_REORIENT DONE
OUT 311.11  ; T_WB_ROTATE FORWARD WORKBIT
; rung 2: Translates workbit to output.
LD 311.11  ; T_WB_ROTATE FORWARD WORKBIT
ANDNOT 2.03  ; T_INPUT_TESTING STATION EMERGENCY HOME
OUT 0.04  ; T_OUTPUT_TURNTABLE ROTATE FORWARD
; rung 3
LD 311.11  ; T_WB_ROTATE FORWARD WORKBIT
ANDNOT 2.03  ; T_INPUT_TESTING STATION EMERGENCY HOME
TIM 106 #0020
; rung 4: When forward rotate has completed, unclamp the two side clamps until realignment push has completed.
LD TIM106  ; T_LENGTH OF FORWARD ROTATE
OR 311.13  ; T_WB_REORIENT UNCLAMP LENGTH PULSE
ANDNOT 311.14  ; T_WB_RESEATING PUSH DONE
ANDNOT 2.03  ; T_INPUT_TESTING STATION EMERGENCY HOME
OUT 311.13  ; T_WB_REORIENT UNCLAMP LENGTH PULSE
; rung 5: When forward rotate has gone off, pull out the alignment clamp until backwards rotate has completed.
LD TIM106  ; T_LENGTH OF FORWARD ROTATE
OR 311.15  ; T_WB_RETRACT ALIGNMENT CLAMP
ANDNOT 2.03  ; T_INPUT_TESTING STATION EMERGENCY HOME
ANDNOT 312.00  ; T_WB_BACKWARDS ROTATION COMPLETE
ANDNOT 311.09  ; T_WB_REORIENT DONE
OUT 311.15  ; T_WB_RETRACT ALIGNMENT CLAMP

